# B&R Automation Studio project pneutrunk_plc
Automation Studio 4.9

## Configuration Config1

CPU X20CP1684, AutomationRuntime B4.93, Build 4.1.2, Safety 0.0, Vc V4.72.5

### Hardware
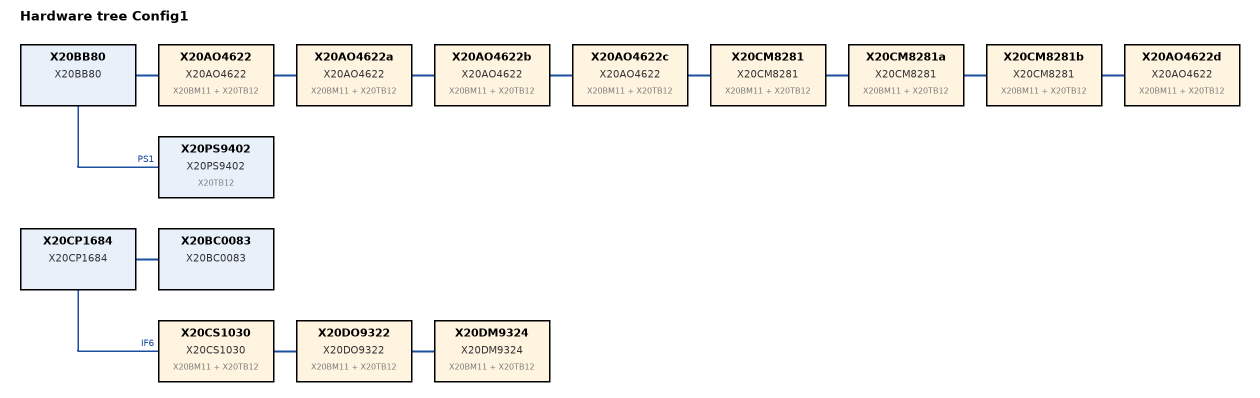
```
X20AO4622 : X20AO4622 v1.3.0.0  [SS1 -> X20TB12a.SS; SL -> X20BM11.SL1]
X20AO4622a : X20AO4622 v1.3.0.0  [SS1 -> X20TB12b.SS; SL -> X20BM11a.SL1]
X20AO4622b : X20AO4622 v1.3.0.0  [SS1 -> X20TB12c.SS; SL -> X20BM11b.SL1]
X20AO4622c : X20AO4622 v1.3.0.0  [SS1 -> X20TB12d.SS; SL -> X20BM11c.SL1]
X20AO4622d : X20AO4622 v1.3.0.0  [SS1 -> X20TB12i.SS; SL -> X20BM11h.SL1]
X20BB80 : X20BB80 v1.1.0.0
X20BC0083 : X20BC0083 v2.14.0.0  [PLK1 -> X20CP1684.IF3 (NodeNumber=1) [Cable Type=PowerlinkCable, Length=10, Version=1.0.0.3]; SL -> X20BB80.SL1]
X20BM11 : X20BM11 v1.1.0.0  [X2X1 -> X20BB80.IF1]
X20BM11a : X20BM11 v1.1.0.0  [X2X1 -> X20BM11.X2X2]
X20BM11b : X20BM11 v1.1.0.0  [X2X1 -> X20BM11a.X2X2]
X20BM11c : X20BM11 v1.1.0.0  [X2X1 -> X20BM11b.X2X2]
X20BM11d : X20BM11 v1.1.0.0  [X2X1 -> X20BM11c.X2X2]
X20BM11e : X20BM11 v1.1.0.0  [X2X1 -> X20BM11d.X2X2]
X20BM11f : X20BM11 v1.1.0.0  [X2X1 -> X20BM11e.X2X2]
X20BM11g : X20BM11 v1.1.0.0  [X2X1 -> X20CP1684.IF6]
X20BM11h : X20BM11 v1.1.0.0  [X2X1 -> X20BM11f.X2X2]
X20BM11i : X20BM11 v1.1.0.0  [X2X1 -> X20BM11g.X2X2]
X20BM11j : X20BM11 v1.1.0.0  [X2X1 -> X20BM11i.X2X2]
X20CM8281 : X20CM8281 v1.4.0.0  [SS1 -> X20TB12e.SS; SL -> X20BM11d.SL1]
X20CM8281a : X20CM8281 v1.4.0.0  [SS1 -> X20TB12f.SS; SL -> X20BM11e.SL1]
X20CM8281b : X20CM8281 v1.4.0.0  [SS1 -> X20TB12g.SS; SL -> X20BM11f.SL1]
X20CP1684 : X20CP1684 v1.5.0.0
  Connector IF2:
    ActivateDevice = 1
    ActivateSnmp = 2
  Connector IF3:
    CycleTime = 500
  ConfigurationID = pneutrunk_Config1
  TimerDeviceType = EPLX2X
  TimerDevice = X20CP1684.IF3
  IdleTaskClass = 4
  TaskClassIdleTime = 2000
  Cyclic1Duration = 2000
  Cyclic1Tolerance = 2000
  Cyclic2Duration = 12000
  Cyclic2Tolerance = 12000
  Cyclic3Duration = 16000
  Cyclic3Tolerance = 16000
  Cyclic4Duration = 50000
  FileDevice1
  FileDeviceName1 = USER
  FileDevicePath1 = USER_PATH
  ActivateDns = 1
  DnsDefaultDomain = br-automation.co.at
  ActivateOpcUa = 1
  OpcUa_Security_AdminRole = Administrators
  OpcUaInformationModels_PV_Version = 1
X20CS1030 : X20CS1030 v1.8.0.0  [SS1 -> X20TB12h.SS; SL -> X20BM11g.SL1]
  Connector IF1:
    Baudrate = 38400
    Parity = N
    DeviceType = RS485
  FunctionModel = StreamCyc1xRS4xx
X20DM9324 : X20DM9324 v1.2.0.0  [SS1 -> X20TB12k.SS; SL -> X20BM11j.SL1]
X20DO9322 : X20DO9322 v1.5.0.0  [SS1 -> X20TB12j.SS; SL -> X20BM11i.SL1]
X20PS9402 : X20PS9402 v1.2.0.0  [SS1 -> X20TB12.SS; PS -> X20BB80.PS1]
X20TB12 : X20TB12 v1.0.0.0
X20TB12a : X20TB12 v1.0.0.0
X20TB12b : X20TB12 v1.0.0.0
X20TB12c : X20TB12 v1.0.0.0
X20TB12d : X20TB12 v1.0.0.0
X20TB12e : X20TB12 v1.0.0.0
X20TB12f : X20TB12 v1.0.0.0
X20TB12g : X20TB12 v1.0.0.0
X20TB12h : X20TB12 v1.0.0.0
X20TB12i : X20TB12 v1.0.0.0
X20TB12j : X20TB12 v1.0.0.0
X20TB12k : X20TB12 v1.0.0.0
```

### IoMap.iom - X20CP1684/IoMap.iom
```iecst
VAR_CONFIG
	::modul.tlak2[5] AT %QW."X20CM8281".AnalogOutput01;
	::modul.tlak3[5] AT %QW."X20CM8281a".AnalogOutput01;
	::modul.tlak1[0] AT %QW."X20AO4622".AnalogOutput01;
	::modul.tlak2[0] AT %QW."X20AO4622".AnalogOutput02;
	::modul.tlak3[0] AT %QW."X20AO4622".AnalogOutput03;
	::modul.tlak1[1] AT %QW."X20AO4622".AnalogOutput04;
	::modul.tlak2[1] AT %QW."X20AO4622a".AnalogOutput01;
	::modul.tlak3[1] AT %QW."X20AO4622a".AnalogOutput02;
	::modul.tlak1[2] AT %QW."X20AO4622a".AnalogOutput03;
	::modul.tlak2[2] AT %QW."X20AO4622a".AnalogOutput04;
	::modul.tlak3[2] AT %QW."X20AO4622b".AnalogOutput01;
	::modul.tlak1[3] AT %QW."X20AO4622b".AnalogOutput02;
	::modul.tlak2[3] AT %QW."X20AO4622b".AnalogOutput03;
	::modul.tlak3[3] AT %QW."X20AO4622b".AnalogOutput04;
	::modul.tlak1[4] AT %QW."X20AO4622c".AnalogOutput01;
	::modul.tlak2[4] AT %QW."X20AO4622c".AnalogOutput02;
	::modul.tlak3[4] AT %QW."X20AO4622c".AnalogOutput03;
	::modul.tlak1[5] AT %QW."X20AO4622c".AnalogOutput04;
	::modul.tlakLinear AT %QW."X20CM8281b".AnalogOutput01;
	::Controller:modull.efektor AT %QX."X20CM8281".DigitalOutput01;
	::modul.tlak2[6] AT %QW."X20AO4622d".AnalogOutput01;
	::modul.tlak3[6] AT %QW."X20AO4622d".AnalogOutput02;
	::modul.tlak1[6] AT %QW."X20AO4622d".AnalogOutput03;
	::zasobnik.ball AT %QX."X20DO9322".DigitalOutput12;
	::zasobnik.ball_piston_sjf AT %QX."X20DO9322".DigitalOutput11;
	::zasobnik.ball_piston AT %QX."X20DO9322".DigitalOutput10;
	::zasobnik.levitovanie AT %QX."X20DO9322".DigitalOutput09;
	::buttons.stropCervenaLED AT %QX."X20DO9322".DigitalOutput08;
	::buttons.startLED AT %QX."X20DO9322".DigitalOutput06;
	::buttons.stopLED AT %QX."X20DO9322".DigitalOutput07;
	::buttons.stropBielaLED AT %QX."X20DO9322".DigitalOutput05;
	::buttons.startButton AT %IX."X20DM9324".DigitalInput01;
	::buttons.stop AT %IX."X20DM9324".DigitalInput02;
	::buttons.centralStop AT %IX."X20DM9324".DigitalInput04;
	::buttons.klucik AT %IX."X20DM9324".DigitalInput03;
END_VAR
```

## Logical view

### Global.typ
```iecst
TYPE
	tlacidla : 	STRUCT
		start : BOOL;
		ros : BOOL;
		stopLED : BOOL;
		stop : BOOL;
		startLED : BOOL;
		startButton : BOOL;
		centralStop : BOOL;
		stropBielaLED : BOOL;
		stropCervenaLED : BOOL;
		klucik : BOOL;
	END_STRUCT;
	automatic : 	STRUCT
		y_desired : ARRAY[0..6]OF INT := [7(0)];
		x_desired : ARRAY[0..6]OF INT := [7(0)];
		linear : INT;
		ball_up : BOOL;
		casovac : BOOL;
		effector : BOOL;
		casovac_uchopenie : BOOL;
		ball_piston : BOOL;
		novyCyklus : TIME := T#1s;
		novyCyklusStart : BOOL;
		trajectoryStart2 : BOOL;
		trajectoryTime2 : TIME := T#6s;
		automatic : BOOL;
		holdPosition : BOOL;
		cas : INT;
		box : INT;
		step_color : INT;
		popcorn : BOOL;
		testFarba : INT;
		loptickyVzasobniku : BOOL := TRUE;
		x_desired_previous : ARRAY[0..6]OF INT;
		y_desired_previous : ARRAY[0..6]OF INT;
		I_konstanta : ARRAY[0..6]OF INT;
		levitacia : BOOL;
	END_STRUCT;
	podavac : 	STRUCT
		levitovanie : BOOL;
		ball_piston_sjf : BOOL;
		ball : BOOL;
		ball_piston : BOOL;
	END_STRUCT;
	identifikacia : 	STRUCT
		p3 : REAL;
		p2 : REAL;
		p1 : REAL;
		vzorka : USINT;
		uhol2 : ARRAY[0..9]OF INT;
		uhol2Priemer : INT;
		uhol1Priemer : INT;
		uhol1 : ARRAY[0..9]OF INT;
		uhol2Stabilny : BOOL;
		uhol1Stabilny : BOOL;
		uhol2Ref : INT;
		uhol1Ref : INT;
		krok : USINT;
		p2Mem : REAL;
		p1Mem : REAL;
		tonStart : BOOL;
		pocetOverenie : USINT := 10;
		spustit : BOOL;
		p3Koniec : BOOL;
		p2Koniec : BOOL;
		p1Koniec : BOOL;
		p3Mem : REAL;
		results : INT;
		switchs : BOOL;
		inkrement : REAL;
		hornyTlak : REAL;
	END_STRUCT;
	packetRS485 : 	STRUCT
		packet : ARRAY[0..9]OF BYTE;
		sendPacketLED : ARRAY[0..5]OF BYTE;
		sendPacketSnimace : ARRAY[0..5]OF BYTE;
		sendPacketFinal : ARRAY[0..5]OF BYTE;
		id : USINT;
	END_STRUCT;
	packetUDP : 	STRUCT
		qDesired : ARRAY[0..40]OF REAL;
		end : INT;
		color : INT;
		step : INT;
		tlak1pos : INT;
		tlak2pos : INT;
		tlak3pos : INT;
		tlak1Full : STRING[80];
		tlak2Full : STRING[80];
		tlak3Full : STRING[80];
		commatlak1 : INT;
		commatlak2 : INT;
		commatlak3 : INT;
		tlak2Desired : ARRAY[0..6]OF REAL;
		tlak1Desired : ARRAY[0..6]OF REAL;
		tlak3Desired : ARRAY[0..6]OF REAL;
		tlak1String : ARRAY[0..6]OF STRING[6];
		tlak2String : ARRAY[0..6]OF STRING[6];
		tlak3String : ARRAY[0..6]OF STRING[6];
		MAX_VALUE : REAL := 32768; (*максимальное значение давления которое может выдержать один модуль*)
	END_STRUCT;
	tlaky : 	STRUCT
		tlak3 : USINT;
		tlak2 : USINT;
		tlak1 : USINT;
	END_STRUCT;
	moduly : 	STRUCT
		uhol2 : ARRAY[0..6]OF REAL := [7(0.0)];
		uhol1 : ARRAY[0..6]OF REAL := [7(0.0)];
		koncak : ARRAY[0..6]OF BOOL;
		led : ARRAY[0..6]OF BOOL;
		uholINT2 : INT;
		uholINT1 : INT;
		tlak1 : ARRAY[0..6]OF INT;
		tlak2 : ARRAY[0..6]OF INT;
		tlak3 : ARRAY[0..6]OF INT;
		tlakLinear : INT;
		uhol_XminusRef : ARRAY[0..6]OF REAL; (*uhol ktory posiela PLC do PC po odpocitani odchylky naklonenia realneho robota*)
		uhol_YminusRef : ARRAY[0..6]OF REAL; (*uhol ktory posiela PLC do PC po odpocitani odchylky naklonenia realneho robota*)
		linearReal : REAL;
		naraz : ARRAY[0..7]OF BOOL;
		narazAktivny : BOOL;
		tlaky : ARRAY[0..3]OF REAL;
	END_STRUCT;
END_TYPE
```

### Global.var
```iecst
VAR
	hranica_upravy_traj : REAL := 2;
	Yellow_tab_ID7 : REAL;
	zasobnik : podavac;
	Yellow_tab_ID6 : REAL;
	I_ON : BOOL;
	Yellow_tab_ID5 : REAL;
	step : INT;
	Yellow_tab_ID4 : REAL;
	Yellow_tab_ID3 : REAL;
	Yellow_tab_ID2 : REAL;
	automatika : automatic;
	Yellow_tab_ID1 : REAL;
	u2 : INT;
	u1 : INT;
	stiffness_ff : REAL;
	result : INT;
	RESET_ID7 : REAL;
	RESET_ID6 : REAL;
	RESET_ID5 : REAL;
	RESET_ID4 : REAL;
	RESET_ID3 : REAL;
	RESET_ID2 : REAL;
	RESET_ID1 : REAL;
	ref_linearny_posun : REAL;
	ref_alfa_y_ID7 : REAL;
	ref_alfa_y_ID6 : REAL;
	ref_alfa_y_ID5 : REAL;
	ref_alfa_y_ID4 : REAL;
	ref_alfa_y_ID3 : REAL;
	ref_alfa_y_ID2 : REAL;
	ref_alfa_y_ID1 : REAL;
	ref_alfa_x_ID7 : REAL;
	ref_alfa_x_ID6 : REAL;
	ref_alfa_x_ID5 : REAL;
	ref_alfa_x_ID4 : REAL;
	ref_alfa_x_ID3 : REAL;
	ref_alfa_x_ID2 : REAL;
	ref_alfa_x_ID1 : REAL;
	q_real : ARRAY[0..12] OF REAL := [0.55,12.58,12.23,7.85,1.23,15.36,17.85,12.05,3.85,3.6,-12.52,10.65,31.28];
	q_desired : ARRAY[0..12] OF REAL;
	pripustna_odchylka_naklonenia : REAL := 0.25;
	poradie_ID7 : REAL;
	poradie_ID6 : REAL;
	poradie_ID5 : REAL;
	poradie_ID4 : REAL;
	poradie_ID3 : REAL;
	poradie_ID2 : REAL;
	poradie_ID1 : REAL;
	packetPos : packetUDP;
	packet485 : packetRS485;
	p3 : REAL;
	p2 : REAL;
	p1 : REAL;
	modul : moduly;
	meranie : identifikacia;
	lin_pressure : REAL;
	I_konstanta_ID7 : REAL;
	I_konstanta_ID6 : REAL;
	I_konstanta_ID5 : REAL;
	I_konstanta_ID4 : REAL;
	I_konstanta_ID3 : REAL;
	I_konstanta_ID2 : REAL;
	cos_test_hodnota2 : REAL;
	cos_test_hodnota1 : REAL;
	I_konstanta_ID1 : REAL;
	Green_tab_ID7 : REAL;
	Green_tab_ID6 : REAL;
	trajectoryStart : BOOL;
	Green_tab_ID5 : REAL;
	Green_tab_ID4 : REAL;
	Green_tab_ID3 : REAL;
	Green_tab_ID2 : REAL;
	Green_tab_ID1 : REAL;
	step_color : INT;
	global_step_udp : INT;
	global_step : INT;
	datagramLength : INT;
	centralStop : BOOL;
	cas_trajektorie : REAL := 100;
	Blue_tab_ID7 : REAL;
	Blue_tab_ID6 : REAL;
	Blue_tab_ID5 : REAL;
	buttons : tlacidla;
	Blue_tab_ID4 : REAL;
	Blue_tab_ID3 : REAL;
	Blue_tab_ID2 : REAL;
	Blue_tab_ID1 : REAL;
	act_alfa_y_ID7 : REAL;
	act_alfa_y_ID6 : REAL;
	act_alfa_y_ID5 : REAL;
	act_alfa_y_ID4 : REAL;
	act_alfa_y_ID3 : REAL;
	act_alfa_y_ID2 : REAL;
	act_alfa_y_ID1 : REAL;
	act_alfa_x_ID7 : REAL;
	act_alfa_x_ID6 : REAL;
	act_alfa_x_ID5 : REAL;
	act_alfa_x_ID4 : REAL;
	act_alfa_x_ID3 : REAL;
	act_alfa_x_ID2 : REAL;
	act_alfa_x_ID1 : REAL;
	clone : INT;
END_VAR
```

### Program Logical/Libraries/regulatory

#### regulator_FF_PI_private.h
```c
/*
 * regulator_FF_PI_private.h
 *
 * Academic License - for use in teaching, academic research, and meeting
 * course requirements at degree granting institutions only.  Not for
 * government, commercial, or other organizational use.
 *
 * Code generation for model "regulator_FF_PI".
 *
 * Model version              : 1.96
 * Simulink Coder version : 9.6 (R2021b) 14-May-2021
 * C source code generated on : Tue Apr  5 15:19:23 2022
 *
 * Target selection: bur_grt.tlc
 * Note: GRT includes extra infrastructure and instrumentation for prototyping
 * Embedded hardware selection: Intel->x86/Pentium
 * Code generation objectives: Unspecified
 * Validation result: Not run
 */

#ifndef RTW_HEADER_regulator_FF_PI_private_h_
#define RTW_HEADER_regulator_FF_PI_private_h_
#include "rtwtypes.h"
#include "multiword_types.h"
#if !defined(rt_VALIDATE_MEMORY)
#define rt_VALIDATE_MEMORY(S, ptr)     if(!(ptr)) {\
 rtmSetErrorStatus(regulator_FF_PI_M, RT_MEMORY_ALLOCATION_ERROR);\
 }
#endif

#if !defined(rt_FREE)
#if !defined(_WIN32)
#define rt_FREE(ptr)                   if((ptr) != (NULL)) {\
 free((ptr));\
 (ptr) = (NULL);\
 }
#else

/* Visual and other windows compilers declare free without const */
#define rt_FREE(ptr)                   if((ptr) != (NULL)) {\
 free((void *)(ptr));\
 (ptr) = (NULL);\
 }
#endif
#endif
#endif                               /* RTW_HEADER_regulator_FF_PI_private_h_ */
```

#### regulator_FF_PI_types.h
```c
/*
 * regulator_FF_PI_types.h
 *
 * Academic License - for use in teaching, academic research, and meeting
 * course requirements at degree granting institutions only.  Not for
 * government, commercial, or other organizational use.
 *
 * Code generation for model "regulator_FF_PI".
 *
 * Model version              : 1.96
 * Simulink Coder version : 9.6 (R2021b) 14-May-2021
 * C source code generated on : Tue Apr  5 15:19:23 2022
 *
 * Target selection: bur_grt.tlc
 * Note: GRT includes extra infrastructure and instrumentation for prototyping
 * Embedded hardware selection: Intel->x86/Pentium
 * Code generation objectives: Unspecified
 * Validation result: Not run
 */

#ifndef RTW_HEADER_regulator_FF_PI_types_h_
#define RTW_HEADER_regulator_FF_PI_types_h_

/* Model Code Variants */

/* Forward declaration for rtModel */

#endif                                 /* RTW_HEADER_regulator_FF_PI_types_h_ */
```

#### PID_co.c
```c
/*
 * PID_co.c
 *
 * Academic License - for use in teaching, academic research, and meeting
 * course requirements at degree granting institutions only.  Not for
 * government, commercial, or other organizational use.
 *
 * Code generation for model "PID_co".
 *
 * Model version              : 1.9
 * Simulink Coder version : 9.6 (R2021b) 14-May-2021
 * C source code generated on : Mon Sep 26 14:43:58 2022
 *
 * Target selection: bur_grt.tlc
 * Note: GRT includes extra infrastructure and instrumentation for prototyping
 * Embedded hardware selection: Intel->x86/Pentium
 * Code generation objectives: Unspecified
 * Validation result: Not run
 */

#include "PID_co.h"
#include "PID_co_private.h"

/* Forward declaration for local functions */
static real32_T PID_co_norm(const real32_T x[4], struct PID_c* inst);

/* Function for MATLAB Function: '<S2>/requested alfa 2 deltaz1' */
static real32_T PID_co_norm(const real32_T x[4], struct PID_c* inst)
{
  real32_T absxk;
  real32_T scale;
  real32_T t;
  real32_T y;
  scale = 1.29246971E-26F;
  absxk = fabsf(x[0]);
  if (absxk > 1.29246971E-26F) {
    y = 1.0F;
    scale = absxk;
  } else {
    t = absxk / 1.29246971E-26F;
    y = t * t;
  }

  absxk = fabsf(x[1]);
  if (absxk > scale) {
    t = scale / absxk;
    y = y * t * t + 1.0F;
    scale = absxk;
  } else {
    t = absxk / scale;
    y += t * t;
  }

  absxk = fabsf(x[2]);
  if (absxk > scale) {
    t = scale / absxk;
    y = y * t * t + 1.0F;
    scale = absxk;
  } else {
    t = absxk / scale;
    y += t * t;
  }

  absxk = fabsf(x[3]);
  if (absxk > scale) {
    t = scale / absxk;
    y = y * t * t + 1.0F;
    scale = absxk;
  } else {
    t = absxk / scale;
    y += t * t;
  }

  return scale * sqrtf(y);
}

/* Model step function */
void PID_co_step(RT_MODEL_PID_co_T *const PID_co_M, struct PID_c* inst)
{
  B_PID_co_T *PID_co_B = PID_co_M->blockIO;
  DW_PID_co_T *PID_co_DW = PID_co_M->dwork;
  real_T Tz23[16];
  real_T Blue0_tmp[4];
  real_T Yellow0_tmp[4];
  real_T A1;
  real_T A2;
  real_T A3;
  real_T rtb_Sum1;
  real_T rtb_Sum2;
  real_T rtb_Sum_j;
  real_T u0;
  int32_T Tz23_tmp;
  int32_T Tz23_tmp_tmp;
  int32_T i;
  int32_T i_0;
  real32_T AlphaY_0[16];
  real32_T HTransform[16];
  real32_T HTransform_tmp_3[16];
  real32_T Tz23_0[16];
  real32_T Blue0_tmp_0[4];
  real32_T Green0_tmp_tmp_0[4];
  real32_T Yellow0_tmp_0[4];
  real32_T Yellow0_tmp_1[4];
  real32_T AlphaX;
  real32_T AlphaY;
  real32_T HTransform_tmp;
  real32_T HTransform_tmp_0;
  int8_T Green0_tmp_tmp[4];
  int8_T HTransform_tmp_1[4];
  int8_T HTransform_tmp_2[4];

  /* S-Function (bur_in): '<Root>/Input1' */
  PID_co_B->Input1 = inst->ref_alfa_x;

  /* S-Function (bur_in): '<Root>/Input2' */
  PID_co_B->Input2 = inst->ref_alfa_y;

  /* S-Function (bur_in): '<Root>/Input3' */
  PID_co_B->Input3 = inst->real_alfa_x;

  /* S-Function (bur_in): '<Root>/Input4' */
  PID_co_B->Input4 = inst->real_alfa_y;

  /* MATLAB Function: '<S2>/requested alfa 2 deltaz1' incorporates:
   *  Constant: '<S2>/Constant1'
   */
  AlphaX = PID_co_B->Input1 * 3.14159274F / 180.0F;
  AlphaY = -PID_co_B->Input2 * 3.14159274F / 180.0F;
  Tz23[2] = 0.0;
  Tz23[6] = 0.0;
  Tz23[10] = 1.0;
  Tz23[14] = 57.5;
  HTransform_tmp = sinf(AlphaY);
  AlphaY = cosf(AlphaY);
  HTransform_tmp_0 = sinf(AlphaX);
  AlphaX = cosf(AlphaX);
  AlphaY_0[0] = AlphaY;
  AlphaY_0[4] = 0.0F;
  AlphaY_0[8] = HTransform_tmp;
  AlphaY_0[12] = 0.0F;
  AlphaY_0[2] = -HTransform_tmp;
  AlphaY_0[6] = 0.0F;
  AlphaY_0[10] = AlphaY;
  AlphaY_0[14] = 0.0F;
  Tz23[0] = 1.0;
  Tz23[1] = 0.0;
  Tz23[3] = 0.0;
  HTransform_tmp_2[0] = 1;
  AlphaY_0[1] = 0.0F;
  AlphaY_0[3] = 0.0F;
  HTransform_tmp_1[0] = 0;
  Tz23[4] = 0.0;
  Tz23[5] = 1.0;
  Tz23[7] = 0.0;
  HTransform_tmp_2[1] = 0;
  AlphaY_0[5] = 1.0F;
  AlphaY_0[7] = 0.0F;
  HTransform_tmp_1[1] = 0;
  Tz23[8] = 0.0;
  Tz23[9] = 0.0;
  Tz23[11] = 0.0;
  HTransform_tmp_2[2] = 0;
  AlphaY_0[9] = 0.0F;
  AlphaY_0[11] = 0.0F;
  HTransform_tmp_1[2] = 0;
  Tz23[12] = 0.0;
  Tz23[13] = 0.0;
  Tz23[15] = 1.0;
  HTransform_tmp_2[3] = 0;
  AlphaY_0[13] = 0.0F;
  AlphaY_0[15] = 1.0F;
  HTransform_tmp_1[3] = 1;
  HTransform_tmp_3[1] = 0.0F;
  HTransform_tmp_3[5] = AlphaX;
  HTransform_tmp_3[9] = -HTransform_tmp_0;
  HTransform_tmp_3[13] = 0.0F;
  HTransform_tmp_3[2] = 0.0F;
  HTransform_tmp_3[6] = HTransform_tmp_0;
  HTransform_tmp_3[10] = AlphaX;
  HTransform_tmp_3[14] = 0.0F;
  for (i = 0; i < 4; i++) {
    for (i_0 = 0; i_0 < 4; i_0++) {
      Tz23_tmp_tmp = i_0 << 2;
      Tz23_tmp = i + Tz23_tmp_tmp;
      Tz23_0[Tz23_tmp] = 0.0F;
      Tz23_0[Tz23_tmp] += AlphaY_0[Tz23_tmp_tmp] * (real32_T)Tz23[i];
      Tz23_0[Tz23_tmp] += AlphaY_0[Tz23_tmp_tmp + 1] * (real32_T)Tz23[i + 4];
      Tz23_0[Tz23_tmp] += AlphaY_0[Tz23_tmp_tmp + 2] * (real32_T)Tz23[i + 8];
      Tz23_0[Tz23_tmp] += AlphaY_0[Tz23_tmp_tmp + 3] * (real32_T)Tz23[i + 12];
    }

    Tz23_tmp_tmp = i << 2;
    HTransform_tmp_3[Tz23_tmp_tmp] = HTransform_tmp_2[i];
    HTransform_tmp_3[Tz23_tmp_tmp + 3] = HTransform_tmp_1[i];
  }

  Green0_tmp_tmp[0] = 85;
  Green0_tmp_tmp[1] = 0;
  Green0_tmp_tmp[2] = 0;
  Green0_tmp_tmp[3] = 1;
  Yellow0_tmp[0] = -42.5;
  Yellow0_tmp[1] = 73.612159321677282;
  Yellow0_tmp[2] = 0.0;
  Yellow0_tmp[3] = 1.0;
  Blue0_tmp[0] = -42.5;
  Blue0_tmp[1] = -73.612159321677282;
  Blue0_tmp[2] = 0.0;
  Blue0_tmp[3] = 1.0;
  for (i = 0; i < 4; i++) {
    for (i_0 = 0; i_0 < 4; i_0++) {
      Tz23_tmp_tmp = i_0 << 2;
      Tz23_tmp = i + Tz23_tmp_tmp;
      AlphaY_0[Tz23_tmp] = 0.0F;
      AlphaY_0[Tz23_tmp] += HTransform_tmp_3[Tz23_tmp_tmp] * Tz23_0[i];
      AlphaY_0[Tz23_tmp] += HTransform_tmp_3[Tz23_tmp_tmp + 1] * Tz23_0[i + 4];
      AlphaY_0[Tz23_tmp] += HTransform_tmp_3[Tz23_tmp_tmp + 2] * Tz23_0[i + 8];
      AlphaY_0[Tz23_tmp] += HTransform_tmp_3[Tz23_tmp_tmp + 3] * Tz23_0[i + 12];
    }

    AlphaX = 0.0F;
    AlphaY = 0.0F;
    HTransform_tmp = 0.0F;
    for (i_0 = 0; i_0 < 4; i_0++) {
      Tz23_tmp_tmp = i_0 << 2;
      Tz23_tmp = i + Tz23_tmp_tmp;
      HTransform[Tz23_tmp] = 0.0F;
      HTransform[Tz23_tmp] += (real32_T)Tz23[Tz23_tmp_tmp] * AlphaY_0[i];
      HTransform[Tz23_tmp] += (real32_T)Tz23[Tz23_tmp_tmp + 1] * AlphaY_0[i + 4];
      HTransform[Tz23_tmp] += (real32_T)Tz23[Tz23_tmp_tmp + 2] * AlphaY_0[i + 8];
      HTransform[Tz23_tmp] += (real32_T)Tz23[Tz23_tmp_tmp + 3] * AlphaY_0[i + 12];
      AlphaX += HTransform[Tz23_tmp] * (real32_T)Green0_tmp_tmp[i_0];
      AlphaY += HTransform[Tz23_tmp] * (real32_T)Yellow0_tmp[i_0];
      HTransform_tmp += HTransform[Tz23_tmp] * (real32_T)Blue0_tmp[i_0];
    }

    Green0_tmp_tmp_0[i] = (real32_T)Green0_tmp_tmp[i] - AlphaX;
    Yellow0_tmp_0[i] = (real32_T)Yellow0_tmp[i] - AlphaY;
    Blue0_tmp_0[i] = (real32_T)Blue0_tmp[i] - HTransform_tmp;
  }

  AlphaX = PID_co_B->Input3 * 3.14159274F / 180.0F;
  AlphaY = -PID_co_B->Input4 * 3.14159274F / 180.0F;
  HTransform_tmp = sinf(AlphaY);
  AlphaY = cosf(AlphaY);
  HTransform_tmp_0 = sinf(AlphaX);
  AlphaX = cosf(AlphaX);
  AlphaY_0[0] = AlphaY;
  AlphaY_0[4] = 0.0F;
  AlphaY_0[8] = HTransform_tmp;
  AlphaY_0[12] = 0.0F;
  AlphaY_0[2] = -HTransform_tmp;
  AlphaY_0[6] = 0.0F;
  AlphaY_0[10] = AlphaY;
  AlphaY_0[14] = 0.0F;
  AlphaY_0[1] = 0.0F;
  AlphaY_0[3] = 0.0F;
  AlphaY_0[5] = 1.0F;
  AlphaY_0[7] = 0.0F;
  AlphaY_0[9] = 0.0F;
  AlphaY_0[11] = 0.0F;
  AlphaY_0[13] = 0.0F;
  AlphaY_0[15] = 1.0F;
  HTransform_tmp_3[1] = 0.0F;
  HTransform_tmp_3[5] = AlphaX;
  HTransform_tmp_3[9] = -HTransform_tmp_0;
  HTransform_tmp_3[13] = 0.0F;
  HTransform_tmp_3[2] = 0.0F;
  HTransform_tmp_3[6] = HTransform_tmp_0;
  HTransform_tmp_3[10] = AlphaX;
  HTransform_tmp_3[14] = 0.0F;
  for (i = 0; i < 4; i++) {
    for (i_0 = 0; i_0 < 4; i_0++) {
      Tz23_tmp_tmp = i_0 << 2;
      Tz23_tmp = i + Tz23_tmp_tmp;
      Tz23_0[Tz23_tmp] = 0.0F;
      Tz23_0[Tz23_tmp] += AlphaY_0[Tz23_tmp_tmp] * (real32_T)Tz23[i];
      Tz23_0[Tz23_tmp] += AlphaY_0[Tz23_tmp_tmp + 1] * (real32_T)Tz23[i + 4];
      Tz23_0[Tz23_tmp] += AlphaY_0[Tz23_tmp_tmp + 2] * (real32_T)Tz23[i + 8];
      Tz23_0[Tz23_tmp] += AlphaY_0[Tz23_tmp_tmp + 3] * (real32_T)Tz23[i + 12];
    }

    Tz23_tmp_tmp = i << 2;
    HTransform_tmp_3[Tz23_tmp_tmp] = HTransform_tmp_2[i];
    HTransform_tmp_3[Tz23_tmp_tmp + 3] = HTransform_tmp_1[i];
  }

  Yellow0_tmp[0] = -42.5;
  Yellow0_tmp[1] = 73.612159321677282;
  Yellow0_tmp[2] = 0.0;
  Yellow0_tmp[3] = 1.0;
  Blue0_tmp[0] = -42.5;
  Blue0_tmp[1] = -73.612159321677282;
  Blue0_tmp[2] = 0.0;
  Blue0_tmp[3] = 1.0;
  for (i = 0; i < 4; i++) {
    for (i_0 = 0; i_0 < 4; i_0++) {
      Tz23_tmp_tmp = i_0 << 2;
      Tz23_tmp = i + Tz23_tmp_tmp;
      AlphaY_0[Tz23_tmp] = 0.0F;
      AlphaY_0[Tz23_tmp] += HTransform_tmp_3[Tz23_tmp_tmp] * Tz23_0[i];
      AlphaY_0[Tz23_tmp] += HTransform_tmp_3[Tz23_tmp_tmp + 1] * Tz23_0[i + 4];
      AlphaY_0[Tz23_tmp] += HTransform_tmp_3[Tz23_tmp_tmp + 2] * Tz23_0[i + 8];
      AlphaY_0[Tz23_tmp] += HTransform_tmp_3[Tz23_tmp_tmp + 3] * Tz23_0[i + 12];
    }

    AlphaX = 0.0F;
    for (i_0 = 0; i_0 < 4; i_0++) {
      Tz23_tmp_tmp = i_0 << 2;
      Tz23_tmp = i + Tz23_tmp_tmp;
      HTransform[Tz23_tmp] = 0.0F;
      HTransform[Tz23_tmp] += (real32_T)Tz23[Tz23_tmp_tmp] * AlphaY_0[i];
      HTransform[Tz23_tmp] += (real32_T)Tz23[Tz23_tmp_tmp + 1] * AlphaY_0[i + 4];
      HTransform[Tz23_tmp] += (real32_T)Tz23[Tz23_tmp_tmp + 2] * AlphaY_0[i + 8];
      HTransform[Tz23_tmp] += (real32_T)Tz23[Tz23_tmp_tmp + 3] * AlphaY_0[i + 12];
      AlphaX += HTransform[Tz23_tmp] * (real32_T)Yellow0_tmp[i_0];
    }

    Yellow0_tmp_1[i] = (real32_T)Yellow0_tmp[i] - AlphaX;
  }

  /* Sum: '<S1>/Sum' incorporates:
   *  Constant: '<S6>/cylinder height'
   *  Constant: '<S8>/cylinder height'
   *  Gain: '<S2>/Gain'
   *  Gain: '<S2>/Gain3'
   *  MATLAB Function: '<S2>/requested alfa 2 deltaz1'
   *  Sum: '<S6>/Sum'
   *  Sum: '<S8>/Sum'
   */
  rtb_Sum_j = (0.001F * PID_co_norm(Yellow0_tmp_1, inst) - 0.115) - (0.001F *
    PID_co_norm(Yellow0_tmp_0, inst) - 0.115);

  /* S-Function (bur_in): '<Root>/Input11' */
  PID_co_B->Input11 = inst->P_parameter;

  /* S-Function (bur_in): '<Root>/Input5' */
  PID_co_B->Input5 = inst->reset_PID_blue;

  /* DiscreteIntegrator: '<S140>/Integrator' */
  if ((PID_co_B->Input5 <= 0.0F) && (PID_co_DW->Integrator_PrevResetState == 1))
  {
    PID_co_DW->Integrator_DSTATE = 0.0;
  }

  /* S-Function (bur_in): '<Root>/Input13' */
  PID_co_B->Input13 = inst->D_parameter;

  /* DiscreteIntegrator: '<S135>/Filter' */
  if ((PID_co_B->Input5 <= 0.0F) && (PID_co_DW->Filter_PrevResetState == 1)) {
    PID_co_DW->Filter_DSTATE = 0.0;
  }

  /* S-Function (bur_in): '<Root>/Input14' */
  PID_co_B->Input14 = inst->N_parameter;

  /* Product: '<S143>/NProd Out' incorporates:
   *  DiscreteIntegrator: '<S135>/Filter'
   *  Product: '<S134>/DProd Out'
   *  Sum: '<S135>/SumD'
   */
  A1 = (rtb_Sum_j * PID_co_B->Input13 - PID_co_DW->Filter_DSTATE) *
    PID_co_B->Input14;

  /* Switch: '<Root>/Switch2' */
  if (PID_co_B->Input5 > 0.0F) {
    /* Sum: '<S149>/Sum' incorporates:
     *  DiscreteIntegrator: '<S140>/Integrator'
     *  Product: '<S145>/PProd Out'
     */
    u0 = (rtb_Sum_j * PID_co_B->Input11 + PID_co_DW->Integrator_DSTATE) + A1;

    /* Saturate: '<S147>/Saturation' */
    if (u0 > 2.0) {
      /* Switch: '<Root>/Switch2' */
      PID_co_B->Switch2 = 2.0F;
    } else if (u0 < -3.0) {
      /* Switch: '<Root>/Switch2' */
      PID_co_B->Switch2 = -3.0F;
    } else {
      /* Switch: '<Root>/Switch2' */
      PID_co_B->Switch2 = (real32_T)u0;
    }

    /* End of Saturate: '<S147>/Saturation' */
  } else {
    /* Switch: '<Root>/Switch2' */
    PID_co_B->Switch2 = 0.0F;
  }

  /* End of Switch: '<Root>/Switch2' */

  /* S-Function (bur_out): '<Root>/Output1' */
  inst->Blue_tab = PID_co_B->Switch2;

  /* MATLAB Function: '<S2>/requested alfa 2 deltaz1' */
  for (i = 0; i < 4; i++) {
    Yellow0_tmp_0[i] = (real32_T)Blue0_tmp[i] - ((HTransform[i + 4] *
      -73.6121597F + HTransform[i] * -42.5F) + HTransform[i + 12]);
  }

  /* Sum: '<S1>/Sum1' incorporates:
   *  Constant: '<S10>/cylinder height'
   *  Constant: '<S7>/cylinder height'
   *  Gain: '<S2>/Gain2'
   *  Gain: '<S2>/Gain5'
   *  MATLAB Function: '<S2>/requested alfa 2 deltaz1'
   *  Sum: '<S10>/Sum'
   *  Sum: '<S7>/Sum'
   */
  rtb_Sum1 = (0.001F * PID_co_norm(Yellow0_tmp_0, inst) - 0.115) - (0.001F *
    PID_co_norm(Blue0_tmp_0, inst) - 0.115);

  /* S-Function (bur_in): '<Root>/Input6' */
  PID_co_B->Input6 = inst->reset_PID_yellow;

  /* DiscreteIntegrator: '<S44>/Integrator' */
  if ((PID_co_B->Input6 <= 0.0F) && (PID_co_DW->Integrator_PrevResetState_m == 1))
  {
    PID_co_DW->Integrator_DSTATE_f = 0.0;
  }

  /* DiscreteIntegrator: '<S39>/Filter' */
  if ((PID_co_B->Input6 <= 0.0F) && (PID_co_DW->Filter_PrevResetState_e == 1)) {
    PID_co_DW->Filter_DSTATE_j = 0.0;
  }

  /* Product: '<S47>/NProd Out' incorporates:
   *  DiscreteIntegrator: '<S39>/Filter'
   *  Product: '<S38>/DProd Out'
   *  Sum: '<S39>/SumD'
   */
  A2 = (rtb_Sum1 * PID_co_B->Input13 - PID_co_DW->Filter_DSTATE_j) *
    PID_co_B->Input14;

  /* Switch: '<Root>/Switch1' */
  if (PID_co_B->Input6 > 0.0F) {
    /* Sum: '<S53>/Sum' incorporates:
     *  DiscreteIntegrator: '<S44>/Integrator'
     *  Product: '<S49>/PProd Out'
     */
    u0 = (rtb_Sum1 * PID_co_B->Input11 + PID_co_DW->Integrator_DSTATE_f) + A2;

    /* Saturate: '<S51>/Saturation' */
    if (u0 > 2.0) {
      /* Switch: '<Root>/Switch1' */
      PID_co_B->Switch1 = 2.0F;
    } else if (u0 < -3.0) {
      /* Switch: '<Root>/Switch1' */
      PID_co_B->Switch1 = -3.0F;
    } else {
      /* Switch: '<Root>/Switch1' */
      PID_co_B->Switch1 = (real32_T)u0;
    }

    /* End of Saturate: '<S51>/Saturation' */
  } else {
    /* Switch: '<Root>/Switch1' */
    PID_co_B->Switch1 = 0.0F;
  }

  /* End of Switch: '<Root>/Switch1' */

  /* S-Function (bur_out): '<Root>/Output2' */
  inst->Yellow_tab = PID_co_B->Switch1;

  /* MATLAB Function: '<S2>/requested alfa 2 deltaz1' */
  for (i = 0; i < 4; i++) {
    Blue0_tmp_0[i] = (real32_T)Green0_tmp_tmp[i] - (HTransform[i] * 85.0F +
      HTransform[i + 12]);
  }

  /* Sum: '<S1>/Sum2' incorporates:
   *  Constant: '<S11>/cylinder height'
   *  Constant: '<S9>/cylinder height'
   *  Gain: '<S2>/Gain1'
   *  Gain: '<S2>/Gain4'
   *  MATLAB Function: '<S2>/requested alfa 2 deltaz1'
   *  Sum: '<S11>/Sum'
   *  Sum: '<S9>/Sum'
   */
  rtb_Sum2 = (0.001F * PID_co_norm(Blue0_tmp_0, inst) - 0.115) - (0.001F * PID_co_norm
    (Green0_tmp_tmp_0, inst) - 0.115);

  /* S-Function (bur_in): '<Root>/Input7' */
  PID_co_B->Input7 = inst->reset_PID_green;

  /* DiscreteIntegrator: '<S92>/Integrator' */
  if ((PID_co_B->Input7 <= 0.0F) && (PID_co_DW->Integrator_PrevResetState_l == 1))
  {
    PID_co_DW->Integrator_DSTATE_h = 0.0;
  }

  /* DiscreteIntegrator: '<S87>/Filter' */
  if ((PID_co_B->Input7 <= 0.0F) && (PID_co_DW->Filter_PrevResetState_k == 1)) {
    PID_co_DW->Filter_DSTATE_m = 0.0;
  }

  /* Product: '<S95>/NProd Out' incorporates:
   *  DiscreteIntegrator: '<S87>/Filter'
   *  Product: '<S86>/DProd Out'
   *  Sum: '<S87>/SumD'
   */
  A3 = (rtb_Sum2 * PID_co_B->Input13 - PID_co_DW->Filter_DSTATE_m) *
    PID_co_B->Input14;

  /* Switch: '<Root>/Switch' */
  if (PID_co_B->Input7 > 0.0F) {
    /* Sum: '<S101>/Sum' incorporates:
     *  DiscreteIntegrator: '<S92>/Integrator'
     *  Product: '<S97>/PProd Out'
     */
    u0 = (rtb_Sum2 * PID_co_B->Input11 + PID_co_DW->Integrator_DSTATE_h) + A3;

    /* Saturate: '<S99>/Saturation' */
    if (u0 > 2.0) {
      /* Switch: '<Root>/Switch' */
      PID_co_B->Switch = 2.0F;
    } else if (u0 < -3.0) {
      /* Switch: '<Root>/Switch' */
      PID_co_B->Switch = -3.0F;
    } else {
      /* Switch: '<Root>/Switch' */
      PID_co_B->Switch = (real32_T)u0;
    }

    /* End of Saturate: '<S99>/Saturation' */
  } else {
    /* Switch: '<Root>/Switch' */
    PID_co_B->Switch = 0.0F;
  }

  /* End of Switch: '<Root>/Switch' */

  /* S-Function (bur_out): '<Root>/Output4' */
  inst->Green_tab = PID_co_B->Switch;

  /* S-Function (bur_in): '<Root>/Input12' */
  PID_co_B->Input12 = inst->I_parameter;

  /* Product: '<S41>/IProd Out' */
  rtb_Sum1 *= PID_co_B->Input12;

  /* Product: '<S89>/IProd Out' */
  rtb_Sum2 *= PID_co_B->Input12;

  /* Product: '<S137>/IProd Out' */
  rtb_Sum_j *= PID_co_B->Input12;

  /* Update for DiscreteIntegrator: '<S140>/Integrator' */
  PID_co_DW->Integrator_DSTATE += 0.002 * rtb_Sum_j;
  if (PID_co_B->Input5 > 0.0F) {
    PID_co_DW->Integrator_PrevResetState = 1;
  } else if (PID_co_B->Input5 < 0.0F) {
    PID_co_DW->Integrator_PrevResetState = -1;
  } else if (PID_co_B->Input5 == 0.0F) {
    PID_co_DW->Integrator_PrevResetState = 0;
  } else {
    PID_co_DW->Integrator_PrevResetState = 2;
  }

  /* End of Update for DiscreteIntegrator: '<S140>/Integrator' */

  /* Update for DiscreteIntegrator: '<S135>/Filter' */
  PID_co_DW->Filter_DSTATE += 0.002 * A1;
  if (PID_co_B->Input5 > 0.0F) {
    PID_co_DW->Filter_PrevResetState = 1;
  } else if (PID_co_B->Input5 < 0.0F) {
    PID_co_DW->Filter_PrevResetState = -1;
  } else if (PID_co_B->Input5 == 0.0F) {
    PID_co_DW->Filter_PrevResetState = 0;
  } else {
    PID_co_DW->Filter_PrevResetState = 2;
  }

  /* End of Update for DiscreteIntegrator: '<S135>/Filter' */

  /* Update for DiscreteIntegrator: '<S44>/Integrator' */
  PID_co_DW->Integrator_DSTATE_f += 0.002 * rtb_Sum1;
  if (PID_co_B->Input6 > 0.0F) {
    PID_co_DW->Integrator_PrevResetState_m = 1;
  } else if (PID_co_B->Input6 < 0.0F) {
    PID_co_DW->Integrator_PrevResetState_m = -1;
  } else if (PID_co_B->Input6 == 0.0F) {
    PID_co_DW->Integrator_PrevResetState_m = 0;
  } else {
    PID_co_DW->Integrator_PrevResetState_m = 2;
  }

  /* End of Update for DiscreteIntegrator: '<S44>/Integrator' */

  /* Update for DiscreteIntegrator: '<S39>/Filter' */
  PID_co_DW->Filter_DSTATE_j += 0.002 * A2;
  if (PID_co_B->Input6 > 0.0F) {
    PID_co_DW->Filter_PrevResetState_e = 1;
  } else if (PID_co_B->Input6 < 0.0F) {
    PID_co_DW->Filter_PrevResetState_e = -1;
  } else if (PID_co_B->Input6 == 0.0F) {
    PID_co_DW->Filter_PrevResetState_e = 0;
  } else {
    PID_co_DW->Filter_PrevResetState_e = 2;
  }

  /* End of Update for DiscreteIntegrator: '<S39>/Filter' */

  /* Update for DiscreteIntegrator: '<S92>/Integrator' */
  PID_co_DW->Integrator_DSTATE_h += 0.002 * rtb_Sum2;
  if (PID_co_B->Input7 > 0.0F) {
    PID_co_DW->Integrator_PrevResetState_l = 1;
  } else if (PID_co_B->Input7 < 0.0F) {
    PID_co_DW->Integrator_PrevResetState_l = -1;
  } else if (PID_co_B->Input7 == 0.0F) {
    PID_co_DW->Integrator_PrevResetState_l = 0;
  } else {
    PID_co_DW->Integrator_PrevResetState_l = 2;
  }

  /* End of Update for DiscreteIntegrator: '<S92>/Integrator' */

  /* Update for DiscreteIntegrator: '<S87>/Filter' */
  PID_co_DW->Filter_DSTATE_m += 0.002 * A3;
  if (PID_co_B->Input7 > 0.0F) {
    PID_co_DW->Filter_PrevResetState_k = 1;
  } else if (PID_co_B->Input7 < 0.0F) {
    PID_co_DW->Filter_PrevResetState_k = -1;
  } else if (PID_co_B->Input7 == 0.0F) {
    PID_co_DW->Filter_PrevResetState_k = 0;
  } else {
    PID_co_DW->Filter_PrevResetState_k = 2;
  }

  /* End of Update for DiscreteIntegrator: '<S87>/Filter' */
}

/* Model initialize function */
void PID_co_initialize(RT_MODEL_PID_co_T *const PID_co_M, struct PID_c* inst)
{
  DW_PID_co_T *PID_co_DW = PID_co_M->dwork;

  /* InitializeConditions for DiscreteIntegrator: '<S140>/Integrator' */
  PID_co_DW->Integrator_DSTATE = 0.0;
  PID_co_DW->Integrator_PrevResetState = 2;

  /* InitializeConditions for DiscreteIntegrator: '<S135>/Filter' */
  PID_co_DW->Filter_DSTATE = 0.0;
  PID_co_DW->Filter_PrevResetState = 2;

  /* InitializeConditions for DiscreteIntegrator: '<S44>/Integrator' */
  PID_co_DW->Integrator_DSTATE_f = 0.0;
  PID_co_DW->Integrator_PrevResetState_m = 2;

  /* InitializeConditions for DiscreteIntegrator: '<S39>/Filter' */
  PID_co_DW->Filter_DSTATE_j = 0.0;
  PID_co_DW->Filter_PrevResetState_e = 2;

  /* InitializeConditions for DiscreteIntegrator: '<S92>/Integrator' */
  PID_co_DW->Integrator_DSTATE_h = 0.0;
  PID_co_DW->Integrator_PrevResetState_l = 2;

  /* InitializeConditions for DiscreteIntegrator: '<S87>/Filter' */
  PID_co_DW->Filter_DSTATE_m = 0.0;
  PID_co_DW->Filter_PrevResetState_k = 2;
}

/* Model terminate function */
void PID_co_terminate(RT_MODEL_PID_co_T * PID_co_M, struct PID_c* inst)
{}

/* Model data allocation function */
void PID_co_initializeMemory(RT_MODEL_PID_co_T* const PID_co_M, struct PID_c * inst)
{  /* states (dwork) */
  {
  }

  {
    B_PID_co_T *PID_co_B = PID_co_M->blockIO;
    DW_PID_co_T *PID_co_DW = PID_co_M->dwork;

    /* block I/O */
    {
      PID_co_B->Input1 = 0.0F;
      PID_co_B->Input2 = 0.0F;
      PID_co_B->Input3 = 0.0F;
      PID_co_B->Input4 = 0.0F;
      PID_co_B->Input11 = 0.0F;
      PID_co_B->Input5 = 0.0F;
      PID_co_B->Input13 = 0.0F;
      PID_co_B->Input14 = 0.0F;
      PID_co_B->Switch2 = 0.0F;
      PID_co_B->Input6 = 0.0F;
      PID_co_B->Switch1 = 0.0F;
      PID_co_B->Input7 = 0.0F;
      PID_co_B->Switch = 0.0F;
      PID_co_B->Input12 = 0.0F;
    }

    /* states (dwork) */
    (void) memset((void *)PID_co_DW, 0,
                  sizeof(DW_PID_co_T));
    PID_co_DW->Integrator_DSTATE = 0.0;
    PID_co_DW->Filter_DSTATE = 0.0;
    PID_co_DW->Integrator_DSTATE_f = 0.0;
    PID_co_DW->Filter_DSTATE_j = 0.0;
    PID_co_DW->Integrator_DSTATE_h = 0.0;
    PID_co_DW->Filter_DSTATE_m = 0.0;
  }

}
```

#### regulator_FF_PI_data.c
```c
/*
 * regulator_FF_PI_data.c
 *
 * Academic License - for use in teaching, academic research, and meeting
 * course requirements at degree granting institutions only.  Not for
 * government, commercial, or other organizational use.
 *
 * Code generation for model "regulator_FF_PI".
 *
 * Model version              : 1.96
 * Simulink Coder version : 9.6 (R2021b) 14-May-2021
 * C source code generated on : Tue Apr  5 15:19:23 2022
 *
 * Target selection: bur_grt.tlc
 * Note: GRT includes extra infrastructure and instrumentation for prototyping
 * Embedded hardware selection: Intel->x86/Pentium
 * Code generation objectives: Unspecified
 * Validation result: Not run
 */

#include "regulator_FF_PI.h"
#include "regulator_FF_PI_private.h"

/* Constant parameters (default storage) */
const ConstP_regulator_FF_PI_T regulator_FF_PI_ConstP = {
  /* Expression: uhol_tlak_pp
   * Referenced by: '<S1>/Constant'
   */
  { 4.94F, 6.03F, 6.83F, 7.62F, 7.57F, 7.83F, 8.5F, 8.01F, 8.67F, 9.42F, 10.08F,
    8.84F, 9.42F, 10.18F, 11.07F, 11.66F, 12.19F, 9.43F, 9.8F, 1.92F, 4.11F,
    2.18F, 0.05F, 5.8F, 4.08F, 2.15F, 7.57F, 5.65F, 3.94F, 2.0F, 9.02F, 7.47F,
    5.55F, 3.76F, 1.85F, 0.05F, 10.5F, 8.76F, 0.0F, 0.0F, 0.0F, 0.0F, 0.0F, 0.0F,
    0.0F, 0.0F, 0.0F, 0.0F, 0.0F, 0.0F, 0.0F, 0.0F, 0.0F, 0.0F, 0.0F, 0.0F, 0.0F,
    0.4F, 0.6F, 0.6F, 0.6F, 0.8F, 0.8F, 0.8F, 1.0F, 1.0F, 1.0F, 1.0F, 1.2F, 1.2F,
    1.2F, 1.2F, 1.2F, 1.2F, 1.4F, 1.4F, 0.0F, 0.0F, 0.2F, 0.4F, 0.0F, 0.2F, 0.4F,
    0.0F, 0.2F, 0.4F, 0.6F, 0.0F, 0.2F, 0.4F, 0.6F, 0.8F, 1.0F, 0.0F, 0.2F, 0.4F,
    0.6F, 0.8F, 1.0F, 0.8F, 1.0F, 1.2F, 1.0F, 1.2F, 1.4F, 1.6F, 1.2F, 1.4F, 1.6F,
    1.8F, 2.0F, 2.2F, 1.4F, 1.6F },

  /* Expression: uhol_tlak_np
   * Referenced by: '<S1>/Constant1'
   */
  { -2.29F, -5.29F, -3.51F, -2.23F, -1.83F, -0.67F, -0.09F, -7.86F, -6.13F,
    -5.25F, -4.82F, -3.77F, -2.62F, -3.19F, -2.25F, -1.56F, -0.05F, -1.71F,
    -1.28F, 1.79F, 1.38F, 2.1F, 0.01F, 4.31F, 2.37F, 6.03F, 1.44F, 1.98F, 0.04F,
    3.93F, 2.36F, 0.51F, 5.79F, 4.43F, 2.73F, 0.67F, 7.65F, 6.1F, 0.4F, 0.6F,
    0.6F, 0.6F, 0.6F, 0.6F, 0.6F, 0.8F, 0.8F, 0.8F, 0.8F, 0.8F, 0.8F, 0.8F, 0.8F,
    0.8F, 0.8F, 0.8F, 0.8F, 0.0F, 0.0F, 0.4F, 0.4F, 0.6F, 0.6F, 0.8F, 0.0F, 0.4F,
    0.4F, 0.6F, 0.6F, 0.6F, 0.8F, 0.8F, 0.8F, 0.8F, 1.0F, 1.0F, 0.0F, 0.0F, 0.0F,
    0.2F, 0.0F, 0.2F, 0.0F, 0.0F, 0.0F, 0.2F, 0.0F, 0.2F, 0.4F, 0.0F, 0.2F, 0.4F,
    0.6F, 0.0F, 0.2F, 0.4F, 0.6F, 1.0F, 1.2F, 1.2F, 1.4F, 1.4F, 0.8F, 1.2F, 1.4F,
    1.4F, 1.6F, 1.8F, 1.6F, 1.8F, 2.0F, 2.2F, 1.8F, 2.0F },

  /* Expression: uhol_tlak_nn
   * Referenced by: '<S1>/Constant2'
   */
  { -1.72F, -1.83F, -0.28F, -1.85F, -0.46F, -4.83F, -3.32F, -2.2F, -0.69F,
    -4.87F, -3.79F, -2.35F, -1.56F, -1.39F, -7.41F, -6.11F, -5.01F, -3.56F,
    -2.32F, -0.54F, -2.15F, -4.45F, -0.45F, -2.72F, -2.12F, -4.46F, -6.89F,
    -8.68F, -0.65F, -2.94F, -4.5F, -6.45F, -2.03F, -1.75F, -4.13F, -6.33F,
    -8.17F, -9.7F, 0.0F, 0.4F, 0.4F, 0.4F, 0.4F, 0.6F, 0.6F, 0.6F, 0.6F, 0.6F,
    0.6F, 0.6F, 0.6F, 0.6F, 0.8F, 0.8F, 0.8F, 0.8F, 0.8F, 0.0F, 0.0F, 0.0F, 0.2F,
    0.2F, 0.0F, 0.0F, 0.0F, 0.0F, 0.2F, 0.2F, 0.2F, 0.2F, 0.4F, 0.0F, 0.0F, 0.0F,
    0.0F, 0.0F, 0.0F, 0.2F, 0.4F, 0.0F, 0.2F, 0.2F, 0.4F, 0.6F, 0.8F, 0.0F, 0.2F,
    0.4F, 0.6F, 0.4F, 0.2F, 0.4F, 0.6F, 0.8F, 1.0F, 0.0F, 0.6F, 0.8F, 0.6F, 0.8F,
    0.8F, 1.0F, 1.2F, 1.4F, 0.8F, 1.0F, 1.2F, 1.4F, 1.4F, 1.0F, 1.2F, 1.4F, 1.6F,
    1.8F },

  /* Expression: uhol_tlak_pn
   * Referenced by: '<S1>/Constant3'
   */
  { 0.31F, 1.68F, 2.8F, 3.65F, 4.88F, 5.33F, 5.98F, 6.5F, 6.89F, 7.36F, 7.72F,
    8.02F, 8.38F, 8.59F, 8.75F, 8.93F, 9.11F, 9.45F, 9.93F, -3.43F, -5.5F,
    -7.74F, -9.49F, -11.38F, -12.88F, -14.21F, -14.98F, -15.71F, -16.11F,
    -16.49F, -17.09F, -17.88F, -18.58F, -18.94F, -19.13F, -19.54F, -19.81F,
    -20.0F, 0.0F, 0.0F, 0.0F, 0.0F, 0.0F, 0.0F, 0.0F, 0.0F, 0.0F, 0.0F, 0.0F,
    0.0F, 0.0F, 0.0F, 0.0F, 0.0F, 0.0F, 0.0F, 0.0F, 0.0F, 0.0F, 0.0F, 0.0F, 0.0F,
    0.0F, 0.0F, 0.0F, 0.0F, 0.0F, 0.0F, 0.0F, 0.0F, 0.0F, 0.0F, 0.0F, 0.0F, 0.0F,
    0.0F, 0.2F, 0.4F, 0.6F, 0.8F, 1.0F, 1.2F, 1.4F, 1.6F, 1.8F, 2.0F, 2.2F, 2.4F,
    2.6F, 2.8F, 3.0F, 3.2F, 3.4F, 3.6F, 3.8F, 0.2F, 0.4F, 0.6F, 0.8F, 1.0F, 1.2F,
    1.4F, 1.6F, 1.8F, 2.0F, 2.2F, 2.4F, 2.6F, 2.8F, 3.0F, 3.2F, 3.4F, 3.6F, 3.8F
  }
};
```

### Program Logical/meranie

#### pneutrunkMeranie.h
```c
/*
 * pneutrunkMeranie.h
 *
 * Academic License - for use in teaching, academic research, and meeting
 * course requirements at degree granting institutions only.  Not for
 * government, commercial, or other organizational use.
 *
 * Code generation for model "pneutrunkMeranie".
 *
 * Model version              : 1.6
 * Simulink Coder version : 9.8 (R2022b) 13-May-2022
 * C source code generated on : Wed May 24 11:04:27 2023
 *
 * Target selection: bur_grt.tlc
 * Note: GRT includes extra infrastructure and instrumentation for prototyping
 * Embedded hardware selection: Intel->x86/Pentium
 * Code generation objectives: Unspecified
 * Validation result: Not run
 */

#ifndef RTW_HEADER_pneutrunkMeranie_h_
#define RTW_HEADER_pneutrunkMeranie_h_
#ifndef pneutrunkMeranie_COMMON_INCLUDES_
#define pneutrunkMeranie_COMMON_INCLUDES_
#include "rtwtypes.h"
#include "simstruc.h"
#include "fixedpoint.h"
#include "dt_info.h"
#include "ext_work.h"
#endif                                 /* pneutrunkMeranie_COMMON_INCLUDES_ */

#include <bur/plctypes.h>

#ifdef _DEFAULT_INCLUDES
 #include <AsDefault.h>
#endif

#include "pneutrunkMeranie_types.h"

#ifndef MIN
#define MIN(a,b)	((a) < (b) ? (a) : (b))
#endif

#ifndef MAX
#define MAX(a,b)	((a) > (b) ? (a) : (b))
#endif

#ifndef AST_ROUND
#define AST_ROUND(x) ((x)>=0?(long long)((x)+0.5):(long long)((x)-0.5))
#endif

#include "rt_defines.h"
#include <string.h>
#include "rt_nonfinite.h"
#include "zero_crossing_types.h"

/* Macros for accessing real-time model data structure */
#ifndef rtmGetBlockIO
#define rtmGetBlockIO(rtm)             ((rtm)->blockIO)
#endif

#ifndef rtmSetBlockIO
#define rtmSetBlockIO(rtm, val)        ((rtm)->blockIO = (val))
#endif

#ifndef rtmGetChecksums
#define rtmGetChecksums(rtm)           ((rtm)->Sizes.checksums)
#endif

#ifndef rtmSetChecksums
#define rtmSetChecksums(rtm, val)      ((rtm)->Sizes.checksums = (val))
#endif

#ifndef rtmGetConstBlockIO
#define rtmGetConstBlockIO(rtm)        ((rtm)->constBlockIO)
#endif

#ifndef rtmSetConstBlockIO
#define rtmSetConstBlockIO(rtm, val)   ((rtm)->constBlockIO = (val))
#endif

#ifndef rtmGetContStateDisabled
#define rtmGetContStateDisabled(rtm)   ((rtm)->contStateDisabled)
#endif

#ifndef rtmSetContStateDisabled
#define rtmSetContStateDisabled(rtm, val) ((rtm)->contStateDisabled = (val))
#endif

#ifndef rtmGetContStates
#define rtmGetContStates(rtm)          ((rtm)->contStates)
#endif

#ifndef rtmSetContStates
#define rtmSetContStates(rtm, val)     ((rtm)->contStates = (val))
#endif

#ifndef rtmGetContTimeOutputInconsistentWithStateAtMajorStepFlag
#define rtmGetContTimeOutputInconsistentWithStateAtMajorStepFlag(rtm) ((rtm)->CTOutputIncnstWithState)
#endif

#ifndef rtmSetContTimeOutputInconsistentWithStateAtMajorStepFlag
#define rtmSetContTimeOutputInconsistentWithStateAtMajorStepFlag(rtm, val) ((rtm)->CTOutputIncnstWithState = (val))
#endif

#ifndef rtmGetCtrlRateMdlRefTiming
#define rtmGetCtrlRateMdlRefTiming(rtm) ()
#endif

#ifndef rtmSetCtrlRateMdlRefTiming
#define rtmSetCtrlRateMdlRefTiming(rtm, val) ()
#endif

#ifndef rtmGetCtrlRateMdlRefTimingPtr
#define rtmGetCtrlRateMdlRefTimingPtr(rtm) ()
#endif

#ifndef rtmSetCtrlRateMdlRefTimingPtr
#define rtmSetCtrlRateMdlRefTimingPtr(rtm, val) ()
#endif

#ifndef rtmGetCtrlRateNumTicksToNextHit
#define rtmGetCtrlRateNumTicksToNextHit(rtm) ()
#endif

#ifndef rtmSetCtrlRateNumTicksToNextHit
#define rtmSetCtrlRateNumTicksToNextHit(rtm, val) ()
#endif

#ifndef rtmGetDataMapInfo
#define rtmGetDataMapInfo(rtm)         ()
#endif

#ifndef rtmSetDataMapInfo
#define rtmSetDataMapInfo(rtm, val)    ()
#endif

#ifndef rtmGetDefaultParam
#define rtmGetDefaultParam(rtm)        ((rtm)->defaultParam)
#endif

#ifndef rtmSetDefaultParam
#define rtmSetDefaultParam(rtm, val)   ((rtm)->defaultParam = (val))
#endif

#ifndef rtmGetDerivCacheNeedsReset
#define rtmGetDerivCacheNeedsReset(rtm) ((rtm)->derivCacheNeedsReset)
#endif

#ifndef rtmSetDerivCacheNeedsReset
#define rtmSetDerivCacheNeedsReset(rtm, val) ((rtm)->derivCacheNeedsReset = (val))
#endif

#ifndef rtmGetDirectFeedThrough
#define rtmGetDirectFeedThrough(rtm)   ((rtm)->Sizes.sysDirFeedThru)
#endif

#ifndef rtmSetDirectFeedThrough
#define rtmSetDirectFeedThrough(rtm, val) ((rtm)->Sizes.sysDirFeedThru = (val))
#endif

#ifndef rtmGetErrorStatusFlag
#define rtmGetErrorStatusFlag(rtm)     ((rtm)->errorStatus)
#endif

#ifndef rtmSetErrorStatusFlag
#define rtmSetErrorStatusFlag(rtm, val) ((rtm)->errorStatus = (val))
#endif

#ifndef rtmGetFinalTime
#define rtmGetFinalTime(rtm)           ((rtm)->Timing.tFinal)
#endif

#ifndef rtmSetFinalTime
#define rtmSetFinalTime(rtm, val)      ((rtm)->Timing.tFinal = (val))
#endif

#ifndef rtmGetFirstInitCondFlag
#define rtmGetFirstInitCondFlag(rtm)   ()
#endif

#ifndef rtmSetFirstInitCondFlag
#define rtmSetFirstInitCondFlag(rtm, val) ()
#endif

#ifndef rtmGetIntgData
#define rtmGetIntgData(rtm)            ()
#endif

#ifndef rtmSetIntgData
#define rtmSetIntgData(rtm, val)       ()
#endif

#ifndef rtmGetMdlRefGlobalRuntimeEventIndices
#define rtmGetMdlRefGlobalRuntimeEventIndices(rtm) ()
#endif

#ifndef rtmSetMdlRefGlobalRuntimeEventIndices
#define rtmSetMdlRefGlobalRuntimeEventIndices(rtm, val) ()
#endif

#ifndef rtmGetMdlRefGlobalTID
#define rtmGetMdlRefGlobalTID(rtm)     ()
#endif

#ifndef rtmSetMdlRefGlobalTID
#define rtmSetMdlRefGlobalTID(rtm, val) ()
#endif

#ifndef rtmGetMdlRefGlobalTimerIndices
#define rtmGetMdlRefGlobalTimerIndices(rtm) ()
#endif

#ifndef rtmSetMdlRefGlobalTimerIndices
#define rtmSetMdlRefGlobalTimerIndices(rtm, val) ()
#endif

#ifndef rtmGetMdlRefTriggerTID
#define rtmGetMdlRefTriggerTID(rtm)    ()
#endif

#ifndef rtmSetMdlRefTriggerTID
#define rtmSetMdlRefTriggerTID(rtm, val) ()
#endif

#ifndef rtmGetModelMappingInfo
#define rtmGetModelMappingInfo(rtm)    ((rtm)->SpecialInfo.mappingInfo)
#endif

#ifndef rtmSetModelMappingInfo
#define rtmSetModelMappingInfo(rtm, val) ((rtm)->SpecialInfo.mappingInfo = (val))
#endif

#ifndef rtmGetModelName
#define rtmGetModelName(rtm)           ((rtm)->modelName)
#endif

#ifndef rtmSetModelName
#define rtmSetModelName(rtm, val)      ((rtm)->modelName = (val))
#endif

#ifndef rtmGetNonInlinedSFcns
#define rtmGetNonInlinedSFcns(rtm)     ()
#endif

#ifndef rtmSetNonInlinedSFcns
#define rtmSetNonInlinedSFcns(rtm, val) ()
#endif

#ifndef rtmGetNumBlockIO
#define rtmGetNumBlockIO(rtm)          ((rtm)->Sizes.numBlockIO)
#endif

#ifndef rtmSetNumBlockIO
#define rtmSetNumBlockIO(rtm, val)     ((rtm)->Sizes.numBlockIO = (val))
#endif

#ifndef rtmGetNumBlockParams
#define rtmGetNumBlockParams(rtm)      ((rtm)->Sizes.numBlockPrms)
#endif

#ifndef rtmSetNumBlockParams
#define rtmSetNumBlockParams(rtm, val) ((rtm)->Sizes.numBlockPrms = (val))
#endif

#ifndef rtmGetNumBlocks
#define rtmGetNumBlocks(rtm)           ((rtm)->Sizes.numBlocks)
#endif

#ifndef rtmSetNumBlocks
#define rtmSetNumBlocks(rtm, val)      ((rtm)->Sizes.numBlocks = (val))
#endif

#ifndef rtmGetNumContStates
#define rtmGetNumContStates(rtm)       ((rtm)->Sizes.numContStates)
#endif

#ifndef rtmSetNumContStates
#define rtmSetNumContStates(rtm, val)  ((rtm)->Sizes.numContStates = (val))
#endif

#ifndef rtmGetNumDWork
#define rtmGetNumDWork(rtm)            ((rtm)->Sizes.numDwork)
#endif

#ifndef rtmSetNumDWork
#define rtmSetNumDWork(rtm, val)       ((rtm)->Sizes.numDwork = (val))
#endif

#ifndef rtmGetNumInputPorts
#define rtmGetNumInputPorts(rtm)       ((rtm)->Sizes.numIports)
#endif

#ifndef rtmSetNumInputPorts
#define rtmSetNumInputPorts(rtm, val)  ((rtm)->Sizes.numIports = (val))
#endif

#ifndef rtmGetNumNonSampledZCs
#define rtmGetNumNonSampledZCs(rtm)    ((rtm)->Sizes.numNonSampZCs)
#endif

#ifndef rtmSetNumNonSampledZCs
#define rtmSetNumNonSampledZCs(rtm, val) ((rtm)->Sizes.numNonSampZCs = (val))
#endif

#ifndef rtmGetNumOutputPorts
#define rtmGetNumOutputPorts(rtm)      ((rtm)->Sizes.numOports)
#endif

#ifndef rtmSetNumOutputPorts
#define rtmSetNumOutputPorts(rtm, val) ((rtm)->Sizes.numOports = (val))
#endif

#ifndef rtmGetNumPeriodicContStates
#define rtmGetNumPeriodicContStates(rtm) ((rtm)->Sizes.numPeriodicContStates)
#endif

#ifndef rtmSetNumPeriodicContStates
#define rtmSetNumPeriodicContStates(rtm, val) ((rtm)->Sizes.numPeriodicContStates = (val))
#endif

#ifndef rtmGetNumSFcnParams
#define rtmGetNumSFcnParams(rtm)       ((rtm)->Sizes.numSFcnPrms)
#endif

#ifndef rtmSetNumSFcnParams
#define rtmSetNumSFcnParams(rtm, val)  ((rtm)->Sizes.numSFcnPrms = (val))
#endif

#ifndef rtmGetNumSFunctions
#define rtmGetNumSFunctions(rtm)       ((rtm)->Sizes.numSFcns)
#endif

#ifndef rtmSetNumSFunctions
#define rtmSetNumSFunctions(rtm, val)  ((rtm)->Sizes.numSFcns = (val))
#endif

#ifndef rtmGetNumSampleTimes
#define rtmGetNumSampleTimes(rtm)      ((rtm)->Sizes.numSampTimes)
#endif

#ifndef rtmSetNumSampleTimes
#define rtmSetNumSampleTimes(rtm, val) ((rtm)->Sizes.numSampTimes = (val))
#endif

#ifndef rtmGetNumU
#define rtmGetNumU(rtm)                ((rtm)->Sizes.numU)
#endif

#ifndef rtmSetNumU
#define rtmSetNumU(rtm, val)           ((rtm)->Sizes.numU = (val))
#endif

#ifndef rtmGetNumY
#define rtmGetNumY(rtm)                ((rtm)->Sizes.numY)
#endif

#ifndef rtmSetNumY
#define rtmSetNumY(rtm, val)           ((rtm)->Sizes.numY = (val))
#endif

#ifndef rtmGetOdeF
#define rtmGetOdeF(rtm)                ()
#endif

#ifndef rtmSetOdeF
#define rtmSetOdeF(rtm, val)           ()
#endif

#ifndef rtmGetOdeY
#define rtmGetOdeY(rtm)                ()
#endif

#ifndef rtmSetOdeY
#define rtmSetOdeY(rtm, val)           ()
#endif

#ifndef rtmGetOffsetTimeArray
#define rtmGetOffsetTimeArray(rtm)     ((rtm)->Timing.offsetTimesArray)
#endif

#ifndef rtmSetOffsetTimeArray
#define rtmSetOffsetTimeArray(rtm, val) ((rtm)->Timing.offsetTimesArray = (val))
#endif

#ifndef rtmGetOffsetTimePtr
#define rtmGetOffsetTimePtr(rtm)       ((rtm)->Timing.offsetTimes)
#endif

#ifndef rtmSetOffsetTimePtr
#define rtmSetOffsetTimePtr(rtm, val)  ((rtm)->Timing.offsetTimes = (val))
#endif

#ifndef rtmGetOptions
#define rtmGetOptions(rtm)             ((rtm)->Sizes.options)
#endif

#ifndef rtmSetOptions
#define rtmSetOptions(rtm, val)        ((rtm)->Sizes.options = (val))
#endif

#ifndef rtmGetParamIsMalloced
#define rtmGetParamIsMalloced(rtm)     ()
#endif

#ifndef rtmSetParamIsMalloced
#define rtmSetParamIsMalloced(rtm, val) ()
#endif

#ifndef rtmGetPath
#define rtmGetPath(rtm)                ((rtm)->path)
#endif

#ifndef rtmSetPath
#define rtmSetPath(rtm, val)           ((rtm)->path = (val))
#endif

#ifndef rtmGetPerTaskSampleHits
#define rtmGetPerTaskSampleHits(rtm)   ()
#endif

#ifndef rtmSetPerTaskSampleHits
#define rtmSetPerTaskSampleHits(rtm, val) ()
#endif

#ifndef rtmGetPerTaskSampleHitsArray
#define rtmGetPerTaskSampleHitsArray(rtm) ((rtm)->Timing.perTaskSampleHitsArray)
#endif

#ifndef rtmSetPerTaskSampleHitsArray
#define rtmSetPerTaskSampleHitsArray(rtm, val) ((rtm)->Timing.perTaskSampleHitsArray = (val))
#endif

#ifndef rtmGetPerTaskSampleHitsPtr
#define rtmGetPerTaskSampleHitsPtr(rtm) ((rtm)->Timing.perTaskSampleHits)
#endif

#ifndef rtmSetPerTaskSampleHitsPtr
#define rtmSetPerTaskSampleHitsPtr(rtm, val) ((rtm)->Timing.perTaskSampleHits = (val))
#endif

#ifndef rtmGetPeriodicContStateIndices
#define rtmGetPeriodicContStateIndices(rtm) ((rtm)->periodicContStateIndices)
#endif

#ifndef rtmSetPeriodicContStateIndices
#define rtmSetPeriodicContStateIndices(rtm, val) ((rtm)->periodicContStateIndices = (val))
#endif

#ifndef rtmGetPeriodicContStateRanges
#define rtmGetPeriodicContStateRanges(rtm) ((rtm)->periodicContStateRanges)
#endif

#ifndef rtmSetPeriodicContStateRanges
#define rtmSetPeriodicContStateRanges(rtm, val) ((rtm)->periodicContStateRanges = (val))
#endif

#ifndef rtmGetPrevZCSigState
#define rtmGetPrevZCSigState(rtm)      ((rtm)->prevZCSigState)
#endif

#ifndef rtmSetPrevZCSigState
#define rtmSetPrevZCSigState(rtm, val) ((rtm)->prevZCSigState = (val))
#endif

#ifndef rtmGetRTWExtModeInfo
#define rtmGetRTWExtModeInfo(rtm)      ((rtm)->extModeInfo)
#endif

#ifndef rtmSetRTWExtModeInfo
#define rtmSetRTWExtModeInfo(rtm, val) ((rtm)->extModeInfo = (val))
#endif

#ifndef rtmGetRTWGeneratedSFcn
#define rtmGetRTWGeneratedSFcn(rtm)    ((rtm)->Sizes.rtwGenSfcn)
#endif

#ifndef rtmSetRTWGeneratedSFcn
#define rtmSetRTWGeneratedSFcn(rtm, val) ((rtm)->Sizes.rtwGenSfcn = (val))
#endif

#ifndef rtmGetRTWLogInfo
#define rtmGetRTWLogInfo(rtm)          ()
#endif

#ifndef rtmSetRTWLogInfo
#define rtmSetRTWLogInfo(rtm, val)     ()
#endif

#ifndef rtmGetRTWRTModelMethodsInfo
#define rtmGetRTWRTModelMethodsInfo(rtm) ()
#endif

#ifndef rtmSetRTWRTModelMethodsInfo
#define rtmSetRTWRTModelMethodsInfo(rtm, val) ()
#endif

#ifndef rtmGetRTWSfcnInfo
#define rtmGetRTWSfcnInfo(rtm)         ((rtm)->sfcnInfo)
#endif

#ifndef rtmSetRTWSfcnInfo
#define rtmSetRTWSfcnInfo(rtm, val)    ((rtm)->sfcnInfo = (val))
#endif

#ifndef rtmGetRTWSolverInfo
#define rtmGetRTWSolverInfo(rtm)       ((rtm)->solverInfo)
#endif

#ifndef rtmSetRTWSolverInfo
#define rtmSetRTWSolverInfo(rtm, val)  ((rtm)->solverInfo = (val))
#endif

#ifndef rtmGetRTWSolverInfoPtr
#define rtmGetRTWSolverInfoPtr(rtm)    ((rtm)->solverInfoPtr)
#endif

#ifndef rtmSetRTWSolverInfoPtr
#define rtmSetRTWSolverInfoPtr(rtm, val) ((rtm)->solverInfoPtr = (val))
#endif

#ifndef rtmGetReservedForXPC
#define rtmGetReservedForXPC(rtm)      ((rtm)->SpecialInfo.xpcData)
#endif

#ifndef rtmSetReservedForXPC
#define rtmSetReservedForXPC(rtm, val) ((rtm)->SpecialInfo.xpcData = (val))
#endif

#ifndef rtmGetRootDWork
#define rtmGetRootDWork(rtm)           ((rtm)->dwork)
#endif

#ifndef rtmSetRootDWork
#define rtmSetRootDWork(rtm, val)      ((rtm)->dwork = (val))
#endif

#ifndef rtmGetSFunctions
#define rtmGetSFunctions(rtm)          ((rtm)->childSfunctions)
#endif

#ifndef rtmSetSFunctions
#define rtmSetSFunctions(rtm, val)     ((rtm)->childSfunctions = (val))
#endif

#ifndef rtmGetSampleHitArray
#define rtmGetSampleHitArray(rtm)      ((rtm)->Timing.sampleHitArray)
#endif

#ifndef rtmSetSampleHitArray
#define rtmSetSampleHitArray(rtm, val) ((rtm)->Timing.sampleHitArray = (val))
#endif

#ifndef rtmGetSampleHitPtr
#define rtmGetSampleHitPtr(rtm)        ((rtm)->Timing.sampleHits)
#endif

#ifndef rtmSetSampleHitPtr
#define rtmSetSampleHitPtr(rtm, val)   ((rtm)->Timing.sampleHits = (val))
#endif

#ifndef rtmGetSampleTimeArray
#define rtmGetSampleTimeArray(rtm)     ((rtm)->Timing.sampleTimesArray)
#endif

#ifndef rtmSetSampleTimeArray
#define rtmSetSampleTimeArray(rtm, val) ((rtm)->Timing.sampleTimesArray = (val))
#endif

#ifndef rtmGetSampleTimePtr
#define rtmGetSampleTimePtr(rtm)       ((rtm)->Timing.sampleTimes)
#endif

#ifndef rtmSetSampleTimePtr
#define rtmSetSampleTimePtr(rtm, val)  ((rtm)->Timing.sampleTimes = (val))
#endif

#ifndef rtmGetSampleTimeTaskIDArray
#define rtmGetSampleTimeTaskIDArray(rtm) ((rtm)->Timing.sampleTimeTaskIDArray)
#endif

#ifndef rtmSetSampleTimeTaskIDArray
#define rtmSetSampleTimeTaskIDArray(rtm, val) ((rtm)->Timing.sampleTimeTaskIDArray = (val))
#endif

#ifndef rtmGetSampleTimeTaskIDPtr
#define rtmGetSampleTimeTaskIDPtr(rtm) ((rtm)->Timing.sampleTimeTaskIDPtr)
#endif

#ifndef rtmSetSampleTimeTaskIDPtr
#define rtmSetSampleTimeTaskIDPtr(rtm, val) ((rtm)->Timing.sampleTimeTaskIDPtr = (val))
#endif

#ifndef rtmGetSelf
#define rtmGetSelf(rtm)                ()
#endif

#ifndef rtmSetSelf
#define rtmSetSelf(rtm, val)           ()
#endif

#ifndef rtmGetSimMode
#define rtmGetSimMode(rtm)             ((rtm)->simMode)
#endif

#ifndef rtmSetSimMode
#define rtmSetSimMode(rtm, val)        ((rtm)->simMode = (val))
#endif

#ifndef rtmGetSimTimeStep
#define rtmGetSimTimeStep(rtm)         ((rtm)->Timing.simTimeStep)
#endif

#ifndef rtmSetSimTimeStep
#define rtmSetSimTimeStep(rtm, val)    ((rtm)->Timing.simTimeStep = (val))
#endif

#ifndef rtmGetStartTime
#define rtmGetStartTime(rtm)           ((rtm)->Timing.tStart)
#endif

#ifndef rtmSetStartTime
#define rtmSetStartTime(rtm, val)      ((rtm)->Timing.tStart = (val))
#endif

#ifndef rtmGetStepSize
#define rtmGetStepSize(rtm)            ((rtm)->Timing.stepSize)
#endif

#ifndef rtmSetStepSize
#define rtmSetStepSize(rtm, val)       ((rtm)->Timing.stepSize = (val))
#endif

#ifndef rtmGetStopRequestedFlag
#define rtmGetStopRequestedFlag(rtm)   ((rtm)->Timing.stopRequestedFlag)
#endif

#ifndef rtmSetStopRequestedFlag
#define rtmSetStopRequestedFlag(rtm, val) ((rtm)->Timing.stopRequestedFlag = (val))
#endif

#ifndef rtmGetTaskCounters
#define rtmGetTaskCounters(rtm)        ()
#endif

#ifndef rtmSetTaskCounters
#define rtmSetTaskCounters(rtm, val)   ()
#endif

#ifndef rtmGetTaskTimeArray
#define rtmGetTaskTimeArray(rtm)       ((rtm)->Timing.tArray)
#endif

#ifndef rtmSetTaskTimeArray
#define rtmSetTaskTimeArray(rtm, val)  ((rtm)->Timing.tArray = (val))
#endif

#ifndef rtmGetTimePtr
#define rtmGetTimePtr(rtm)             ((rtm)->Timing.t)
#endif

#ifndef rtmSetTimePtr
#define rtmSetTimePtr(rtm, val)        ((rtm)->Timing.t = (val))
#endif

#ifndef rtmGetTimingData
#define rtmGetTimingData(rtm)          ((rtm)->Timing.timingData)
#endif

#ifndef rtmSetTimingData
#define rtmSetTimingData(rtm, val)     ((rtm)->Timing.timingData = (val))
#endif

#ifndef rtmGetU
#define rtmGetU(rtm)                   ((rtm)->inputs)
#endif

#ifndef rtmSetU
#define rtmSetU(rtm, val)              ((rtm)->inputs = (val))
#endif

#ifndef rtmGetVarNextHitTimesListPtr
#define rtmGetVarNextHitTimesListPtr(rtm) ((rtm)->Timing.varNextHitTimesList)
#endif

#ifndef rtmSetVarNextHitTimesListPtr
#define rtmSetVarNextHitTimesListPtr(rtm, val) ((rtm)->Timing.varNextHitTimesList = (val))
#endif

#ifndef rtmGetY
#define rtmGetY(rtm)                   ((rtm)->outputs)
#endif

#ifndef rtmSetY
#define rtmSetY(rtm, val)              ((rtm)->outputs = (val))
#endif

#ifndef rtmGetZCCacheNeedsReset
#define rtmGetZCCacheNeedsReset(rtm)   ((rtm)->zCCacheNeedsReset)
#endif

#ifndef rtmSetZCCacheNeedsReset
#define rtmSetZCCacheNeedsReset(rtm, val) ((rtm)->zCCacheNeedsReset = (val))
#endif

#ifndef rtmGetZCSignalValues
#define rtmGetZCSignalValues(rtm)      ((rtm)->zcSignalValues)
#endif

#ifndef rtmSetZCSignalValues
#define rtmSetZCSignalValues(rtm, val) ((rtm)->zcSignalValues = (val))
#endif

#ifndef rtmGet_TimeOfLastOutput
#define rtmGet_TimeOfLastOutput(rtm)   ((rtm)->Timing.timeOfLastOutput)
#endif

#ifndef rtmSet_TimeOfLastOutput
#define rtmSet_TimeOfLastOutput(rtm, val) ((rtm)->Timing.timeOfLastOutput = (val))
#endif

#ifndef rtmGetdX
#define rtmGetdX(rtm)                  ((rtm)->derivs)
#endif

#ifndef rtmSetdX
#define rtmSetdX(rtm, val)             ((rtm)->derivs = (val))
#endif

#ifndef rtmGettimingBridge
#define rtmGettimingBridge(rtm)        ()
#endif

#ifndef rtmSettimingBridge
#define rtmSettimingBridge(rtm, val)   ()
#endif

#ifndef rtmGetChecksumVal
#define rtmGetChecksumVal(rtm, idx)    ((rtm)->Sizes.checksums[idx])
#endif

#ifndef rtmSetChecksumVal
#define rtmSetChecksumVal(rtm, idx, val) ((rtm)->Sizes.checksums[idx] = (val))
#endif

#ifndef rtmGetDWork
#define rtmGetDWork(rtm, idx)          ((rtm)->dwork[idx])
#endif

#ifndef rtmSetDWork
#define rtmSetDWork(rtm, idx, val)     ((rtm)->dwork[idx] = (val))
#endif

#ifndef rtmGetOffsetTime
#define rtmGetOffsetTime(rtm, idx)     ((rtm)->Timing.offsetTimes[idx])
#endif

#ifndef rtmSetOffsetTime
#define rtmSetOffsetTime(rtm, idx, val) ((rtm)->Timing.offsetTimes[idx] = (val))
#endif

#ifndef rtmGetSFunction
#define rtmGetSFunction(rtm, idx)      ((rtm)->childSfunctions[idx])
#endif

#ifndef rtmSetSFunction
#define rtmSetSFunction(rtm, idx, val) ((rtm)->childSfunctions[idx] = (val))
#endif

#ifndef rtmGetSampleTime
#define rtmGetSampleTime(rtm, idx)     ((rtm)->Timing.sampleTimes[idx])
#endif

#ifndef rtmSetSampleTime
#define rtmSetSampleTime(rtm, idx, val) ((rtm)->Timing.sampleTimes[idx] = (val))
#endif

#ifndef rtmGetSampleTimeTaskID
#define rtmGetSampleTimeTaskID(rtm, idx) ((rtm)->Timing.sampleTimeTaskIDPtr[idx])
#endif

#ifndef rtmSetSampleTimeTaskID
#define rtmSetSampleTimeTaskID(rtm, idx, val) ((rtm)->Timing.sampleTimeTaskIDPtr[idx] = (val))
#endif

#ifndef rtmGetVarNextHitTimeList
#define rtmGetVarNextHitTimeList(rtm, idx) ((rtm)->Timing.varNextHitTimesList[idx])
#endif

#ifndef rtmSetVarNextHitTimeList
#define rtmSetVarNextHitTimeList(rtm, idx, val) ((rtm)->Timing.varNextHitTimesList[idx] = (val))
#endif

#ifndef rtmIsContinuousTask
#define rtmIsContinuousTask(rtm, tid)  0
#endif

#ifndef rtmGetErrorStatus
#define rtmGetErrorStatus(rtm)         ((rtm)->errorStatus)
#endif

#ifndef rtmSetErrorStatus
#define rtmSetErrorStatus(rtm, val)    ((rtm)->errorStatus = (val))
#endif

#ifndef rtmIsSampleHit
#define rtmIsSampleHit(rtm, sti, tid)  ((rtm)->Timing.sampleHits[(rtm)->Timing.sampleTimeTaskIDPtr[sti]])
#endif

#ifndef rtmGetStopRequested
#define rtmGetStopRequested(rtm)       ((rtm)->Timing.stopRequestedFlag)
#endif

#ifndef rtmSetStopRequested
#define rtmSetStopRequested(rtm, val)  ((rtm)->Timing.stopRequestedFlag = (val))
#endif

#ifndef rtmGetStopRequestedPtr
#define rtmGetStopRequestedPtr(rtm)    (&((rtm)->Timing.stopRequestedFlag))
#endif

#ifndef rtmGetT
#define rtmGetT(rtm)                   (rtmGetTPtr((rtm))[0])
#endif

#ifndef rtmSetT
#define rtmSetT(rtm, val)                                        /* Do Nothing */
#endif

#ifndef rtmGetTFinal
#define rtmGetTFinal(rtm)              ((rtm)->Timing.tFinal)
#endif

#ifndef rtmSetTFinal
#define rtmSetTFinal(rtm, val)         ((rtm)->Timing.tFinal = (val))
#endif

#ifndef rtmGetTPtr
#define rtmGetTPtr(rtm)                ((rtm)->Timing.t)
#endif

#ifndef rtmSetTPtr
#define rtmSetTPtr(rtm, val)           ((rtm)->Timing.t = (val))
#endif

#ifndef rtmGetTStart
#define rtmGetTStart(rtm)              ((rtm)->Timing.tStart)
#endif

#ifndef rtmSetTStart
#define rtmSetTStart(rtm, val)         ((rtm)->Timing.tStart = (val))
#endif

#ifndef rtmGetTaskTime
#define rtmGetTaskTime(rtm, sti)       (rtmGetTPtr((rtm))[(rtm)->Timing.sampleTimeTaskIDPtr[sti]])
#endif

#ifndef rtmSetTaskTime
#define rtmSetTaskTime(rtm, sti, val)  (rtmGetTPtr((rtm))[sti] = (val))
#endif

#ifndef rtmGetTimeOfLastOutput
#define rtmGetTimeOfLastOutput(rtm)    ((rtm)->Timing.timeOfLastOutput)
#endif

#ifdef rtmGetRTWSolverInfo
#undef rtmGetRTWSolverInfo
#endif

#define rtmGetRTWSolverInfo(rtm)       &((rtm)->solverInfo)

/* Definition for use in the target main file */
#define pneutrunkMeranie_rtModel       RT_MODEL_pneutrunkMeranie_T

/* Block signals (default storage) */
typedef struct {
  real32_T Input;                      /* '<Root>/Input' */
  real32_T Input1;                     /* '<Root>/Input1' */
  real32_T Input2;                     /* '<Root>/Input2' */
  int16_T Input3;                      /* '<Root>/Input3' */
  int16_T Input4;                      /* '<Root>/Input4' */
  int16_T Input5;                      /* '<Root>/Input5' */
} B_pneutrunkMeranie_T;

/* Block states (default storage) for system '<Root>' */
typedef struct {
  struct {
    void *LoggedData;
  } ToWorkspace_PWORK;                 /* '<Root>/To Workspace' */

  struct {
    void *LoggedData;
  } ToWorkspace5_PWORK;                /* '<Root>/To Workspace5' */

  struct {
    void *LoggedData;
  } ToWorkspace4_PWORK;                /* '<Root>/To Workspace4' */

  struct {
    void *LoggedData;
  } ToWorkspace3_PWORK;                /* '<Root>/To Workspace3' */

  struct {
    void *LoggedData;
  } ToWorkspace1_PWORK;                /* '<Root>/To Workspace1' */

  struct {
    void *LoggedData;
  } ToWorkspace2_PWORK;                /* '<Root>/To Workspace2' */
} DW_pneutrunkMeranie_T;

/* Backward compatible GRT Identifiers */
#define rtB                            pneutrunkMeranie_B
#define BlockIO                        B_pneutrunkMeranie_T
#define rtDWork                        pneutrunkMeranie_DW
#define D_Work                         DW_pneutrunkMeranie_T

/* Real-time Model Data Structure */
struct tag_RTM_pneutrunkMeranie_T {
  const char_T *path;
  const char_T *modelName;
  struct SimStruct_tag * *childSfunctions;
  const char_T *errorStatus;
  SS_SimMode simMode;
  RTWExtModeInfo *extModeInfo;
  RTWSolverInfo solverInfo;
  RTWSolverInfo *solverInfoPtr;
  void *sfcnInfo;
  void *blockIO;
  const void *constBlockIO;
  void *defaultParam;
  ZCSigState *prevZCSigState;
  real_T *contStates;
  int_T *periodicContStateIndices;
  real_T *periodicContStateRanges;
  real_T *derivs;
  void *zcSignalValues;
  void *inputs;
  void *outputs;
  boolean_T *contStateDisabled;
  boolean_T zCCacheNeedsReset;
  boolean_T derivCacheNeedsReset;
  boolean_T CTOutputIncnstWithState;
  void *dwork;

  /*
   * Sizes:
   * The following substructure contains sizes information
   * for many of the model attributes such as inputs, outputs,
   * dwork, sample times, etc.
   */
  struct {
    uint32_T checksums[4];
    uint32_T options;
    int_T numContStates;
    int_T numPeriodicContStates;
    int_T numU;
    int_T numY;
    int_T numSampTimes;
    int_T numBlocks;
    int_T numBlockIO;
    int_T numBlockPrms;
    int_T numDwork;
    int_T numSFcnPrms;
    int_T numSFcns;
    int_T numIports;
    int_T numOports;
    int_T numNonSampZCs;
    int_T sysDirFeedThru;
    int_T rtwGenSfcn;
  } Sizes;

  /*
   * SpecialInfo:
   * The following substructure contains special information
   * related to other components that are dependent on RTW.
   */
  struct {
    const void *mappingInfo;
    void *xpcData;
  } SpecialInfo;

  /*
   * Timing:
   * The following substructure contains information regarding
   * the timing information for the model.
   */
  struct {
    time_T stepSize;
    uint32_T clockTick0;
    uint32_T clockTickH0;
    time_T stepSize0;
    time_T tStart;
    time_T tFinal;
    time_T timeOfLastOutput;
    void *timingData;
    real_T *varNextHitTimesList;
    SimTimeStep simTimeStep;
    boolean_T stopRequestedFlag;
    time_T *sampleTimes;
    time_T *offsetTimes;
    int_T *sampleTimeTaskIDPtr;
    int_T *sampleHits;
    int_T *perTaskSampleHits;
    time_T *t;
    time_T sampleTimesArray[1];
    time_T offsetTimesArray[1];
    int_T sampleTimeTaskIDArray[1];
    int_T sampleHitArray[1];
    int_T perTaskSampleHitsArray[1];
    time_T tArray[1];
  } Timing;
};

/* Block signals (default storage) */
extern B_pneutrunkMeranie_T pneutrunkMeranie_B;

/* Block states (default storage) */
extern DW_pneutrunkMeranie_T pneutrunkMeranie_DW;

/* Model entry point functions */
extern void pneutrunkMeranie_initialize(void);
extern void pneutrunkMeranie_output(void);
extern void pneutrunkMeranie_update(void);
extern void pneutrunkMeranie_terminate(void);

/*====================*
 * External functions *
 *====================*/
extern pneutrunkMeranie_rtModel *pneutrunkMeranie(void);
extern void MdlInitializeSizes(void);
extern void MdlInitializeSampleTimes(void);
extern void MdlInitialize(void);
extern void MdlStart(void);
extern void MdlOutputs(int_T tid);
extern void MdlUpdate(int_T tid);
extern void MdlTerminate(void);

/* Real-time Model object */
extern RT_MODEL_pneutrunkMeranie_T *const pneutrunkMeranie_M;

/*-
 * The generated code includes comments that allow you to trace directly
 * back to the appropriate location in the model.  The basic format
 * is <system>/block_name, where system is the system number (uniquely
 * assigned by Simulink) and block_name is the name of the block.
 *
 * Use the MATLAB hilite_system command to trace the generated code back
 * to the model.  For example,
 *
 * hilite_system('<S3>')    - opens system 3
 * hilite_system('<S3>/Kp') - opens and selects block Kp which resides in S3
 *
 * Here is the system hierarchy for this model
 *
 * '<Root>' : 'pneutrunkMeranie'
 */
#endif                                 /* RTW_HEADER_pneutrunkMeranie_h_ */
```

#### rtGetInf.h
```c
/*
 * rtGetInf.h
 *
 * Academic License - for use in teaching, academic research, and meeting
 * course requirements at degree granting institutions only.  Not for
 * government, commercial, or other organizational use.
 *
 * Code generation for model "pneutrunkMeranie".
 *
 * Model version              : 1.6
 * Simulink Coder version : 9.8 (R2022b) 13-May-2022
 * C source code generated on : Wed May 24 11:04:27 2023
 *
 * Target selection: bur_grt.tlc
 * Note: GRT includes extra infrastructure and instrumentation for prototyping
 * Embedded hardware selection: Intel->x86/Pentium
 * Code generation objectives: Unspecified
 * Validation result: Not run
 */

#ifndef RTW_HEADER_rtGetInf_h_
#define RTW_HEADER_rtGetInf_h_
#include "rtwtypes.h"

extern real_T rtGetInf(void);
extern real32_T rtGetInfF(void);
extern real_T rtGetMinusInf(void);
extern real32_T rtGetMinusInfF(void);

#endif                                 /* RTW_HEADER_rtGetInf_h_ */
```

#### rtGetNaN.c
```c
/*
 * rtGetNaN.c
 *
 * Academic License - for use in teaching, academic research, and meeting
 * course requirements at degree granting institutions only.  Not for
 * government, commercial, or other organizational use.
 *
 * Code generation for model "pneutrunkMeranie".
 *
 * Model version              : 1.6
 * Simulink Coder version : 9.8 (R2022b) 13-May-2022
 * C source code generated on : Wed May 24 11:04:27 2023
 *
 * Target selection: bur_grt.tlc
 * Note: GRT includes extra infrastructure and instrumentation for prototyping
 * Embedded hardware selection: Intel->x86/Pentium
 * Code generation objectives: Unspecified
 * Validation result: Not run
 */

#include "rtwtypes.h"
#include "rtGetNaN.h"
#include <stddef.h>
#include "rt_nonfinite.h"
#define NumBitsPerChar                 8U

/*
 * Initialize rtNaN needed by the generated code.
 * NaN is initialized as non-signaling. Assumes IEEE.
 */
real_T rtGetNaN(void)
{
  size_t bitsPerReal = sizeof(real_T) * (NumBitsPerChar);
  real_T nan = 0.0;
  if (bitsPerReal == 32U) {
    nan = rtGetNaNF();
  } else {
    uint16_T one = 1U;
    enum {
      LittleEndian,
      BigEndian
    } machByteOrder = (*((uint8_T *) &one) == 1U) ? LittleEndian : BigEndian;
    switch (machByteOrder) {
     case LittleEndian:
      {
        union {
          LittleEndianIEEEDouble bitVal;
          real_T fltVal;
        } tmpVal;

        tmpVal.bitVal.words.wordH = 0xFFF80000U;
        tmpVal.bitVal.words.wordL = 0x00000000U;
        nan = tmpVal.fltVal;
        break;
      }

     case BigEndian:
      {
        union {
          BigEndianIEEEDouble bitVal;
          real_T fltVal;
        } tmpVal;

        tmpVal.bitVal.words.wordH = 0x7FFFFFFFU;
        tmpVal.bitVal.words.wordL = 0xFFFFFFFFU;
        nan = tmpVal.fltVal;
        break;
      }
    }
  }

  return nan;
}

/*
 * Initialize rtNaNF needed by the generated code.
 * NaN is initialized as non-signaling. Assumes IEEE.
 */
real32_T rtGetNaNF(void)
{
  IEEESingle nanF = { { 0.0F } };

  uint16_T one = 1U;
  enum {
    LittleEndian,
    BigEndian
  } machByteOrder = (*((uint8_T *) &one) == 1U) ? LittleEndian : BigEndian;
  switch (machByteOrder) {
   case LittleEndian:
    {
      nanF.wordL.wordLuint = 0xFFC00000U;
      break;
    }

   case BigEndian:
    {
      nanF.wordL.wordLuint = 0x7FFFFFFFU;
      break;
    }
  }

  return nanF.wordL.wordLreal;
}
```

#### task_properties.txt
```
For manual assignment to hardware configuration please
add the following additional include directories:

\Logical\MATLAB_includes\R2022b\

And the following additional build options:

-lm -DMODEL=pneutrunkMeranie -DNUMST=1 -DNCSTATES=0 -DHAVESTDIO -DRT -DUSE_RTMODEL -DEXT_MODE -DEXTMODE_STATIC -DEXTMODE_STATIC_SIZE=1000000 -DON_TARGET_WAIT_FOR_START=0 -DCLASSIC_INTERFACE=1 -DALLOCATIONFCN=0 -DTID01EQ=0 -DMAT_FILE=0 -DONESTEPFCN=0 -DTERMFCN=1 -DMULTI_INSTANCE_CODE=0 -DINTEGER_CODE=0 -DMT=0
```

### Program Logical/solo_reg
